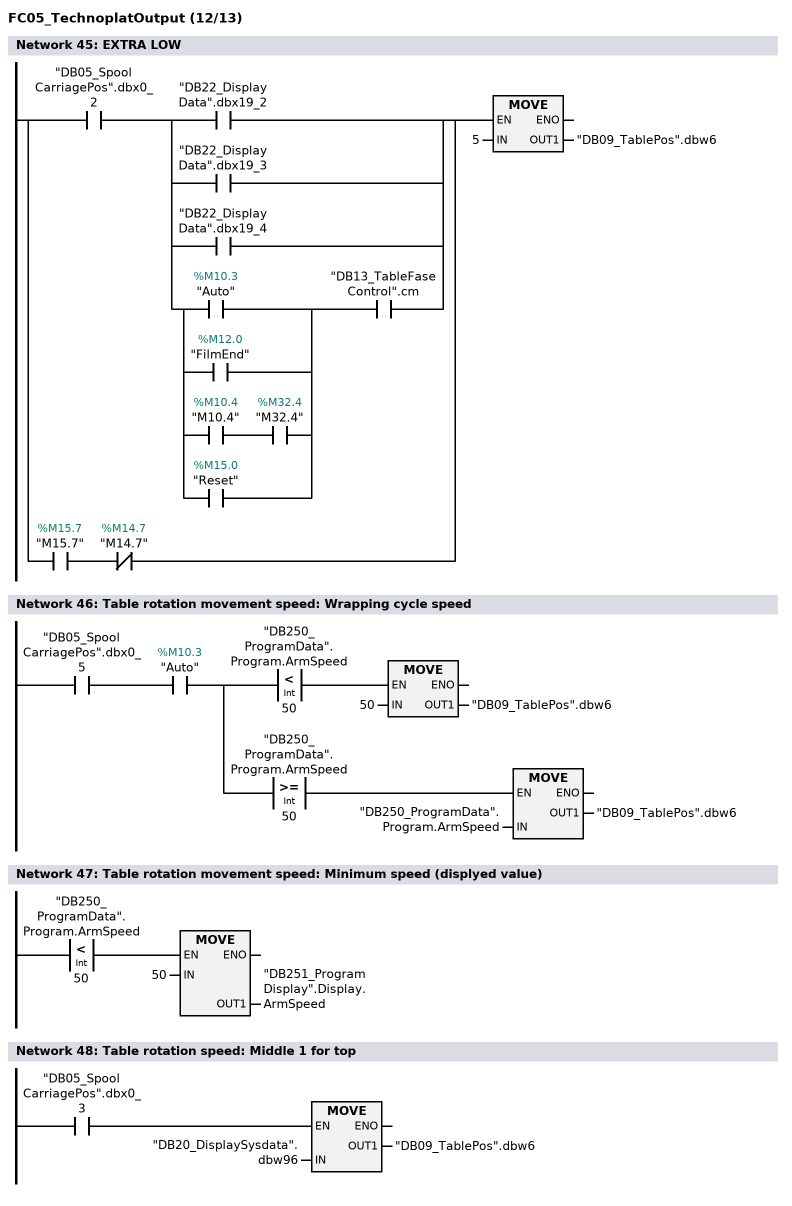
   RUNG wire#powerrail
      Contact( "DB05_SpoolCarriagePos".dbx0_2 )
      wire#w1
      Contact( "DB22_DisplayData".dbx19_2 )
      wire#w2
      { S7_GenerateENO := "TRUE" } Move(in := 5, out1 => "DB09_TablePos".dbw6)
   END_RUNG
   RUNG wire#w1
      Contact( "DB22_DisplayData".dbx19_3 )
   END_RUNG wire#w2
   RUNG wire#w1
      Contact( "DB22_DisplayData".dbx19_4 )
   END_RUNG wire#w2
   RUNG wire#w1
      Contact( "Auto" )
      wire#w3
      Contact( "DB13_TableFaseControl".cm )
   END_RUNG wire#w2
   RUNG wire#w1
      Contact( "FilmEnd" )
   END_RUNG wire#w3
   RUNG wire#w1
      Contact( "M10.4" )
      Contact( "M32.4" )
   END_RUNG wire#w3
   RUNG wire#w1
      Contact( "Reset" )
   END_RUNG wire#w3
   RUNG wire#powerrail
      Contact( "M15.7" )
      I_Contact( "M14.7" )
   END_RUNG wire#w2
   // the same network as SCL:
   IF ("DB05_SpoolCarriagePos".dbx0_2 AND ("DB22_DisplayData".dbx19_2 OR "DB22_DisplayData".dbx19_3 OR "DB22_DisplayData".dbx19_4 OR (("Auto" OR "FilmEnd" OR ("M10.4" AND "M32.4") OR "Reset") AND "DB13_TableFaseControl".cm))) OR ("M15.7" AND NOT "M14.7") THEN
       "DB09_TablePos".dbw6 := 5;
   END_IF;
END_REGION

REGION Network 46: Table rotation movement speed: Wrapping cycle speed
   RUNG wire#powerrail
      Contact( "DB05_SpoolCarriagePos".dbx0_5 )
      Contact( "Auto" )
      wire#w1
      { S7_Templates := "SrcType := Int" } LT_Contact(in1 := "DB250_ProgramData".Program.ArmSpeed, in2 := 50)
      { S7_GenerateENO := "TRUE" } Move(in := 50, out1 => "DB09_TablePos".dbw6)
   END_RUNG
   RUNG wire#w1
      { S7_Templates := "SrcType := Int" } GE_Contact(in1 := "DB250_ProgramData".Program.ArmSpeed, in2 := 50)
      { S7_GenerateENO := "TRUE" } Move(in := "DB250_ProgramData".Program.ArmSpeed, out1 => "DB09_TablePos".dbw6)
   END_RUNG
   // the same network as SCL:
   #_w1 := "DB05_SpoolCarriagePos".dbx0_5 AND "Auto";
   IF #_w1 AND ("DB250_ProgramData".Program.ArmSpeed < 50) THEN "DB09_TablePos".dbw6 := 50; END_IF;
   IF #_w1 AND ("DB250_ProgramData".Program.ArmSpeed >= 50) THEN
       "DB09_TablePos".dbw6 := "DB250_ProgramData".Program.ArmSpeed;
   END_IF;
END_REGION

REGION Network 47: Table rotation movement speed: Minimum speed (displyed value)
   RUNG wire#powerrail
      { S7_Templates := "SrcType := Int" } LT_Contact(in1 := "DB250_ProgramData".Program.ArmSpeed, in2 := 50)
      { S7_GenerateENO := "TRUE" } Move(in := 50, out1 => "DB251_ProgramDisplay".Display.ArmSpeed)
   END_RUNG
   // the same network as SCL:
   IF "DB250_ProgramData".Program.ArmSpeed < 50 THEN "DB251_ProgramDisplay".Display.ArmSpeed := 50; END_IF;
END_REGION

REGION Network 48: Table rotation speed: Middle 1 for top
   RUNG wire#powerrail
      Contact( "DB05_SpoolCarriagePos".dbx0_3 )
      { S7_GenerateENO := "TRUE" } Move(in := "DB20_DisplaySysdata".dbw96, out1 => "DB09_TablePos".dbw6)
   END_RUNG
   // the same network as SCL:
   IF "DB05_SpoolCarriagePos".dbx0_3 THEN "DB09_TablePos".dbw6 := "DB20_DisplaySysdata".dbw96; END_IF;
END_REGION

REGION Network 49: table rotation movement speed range
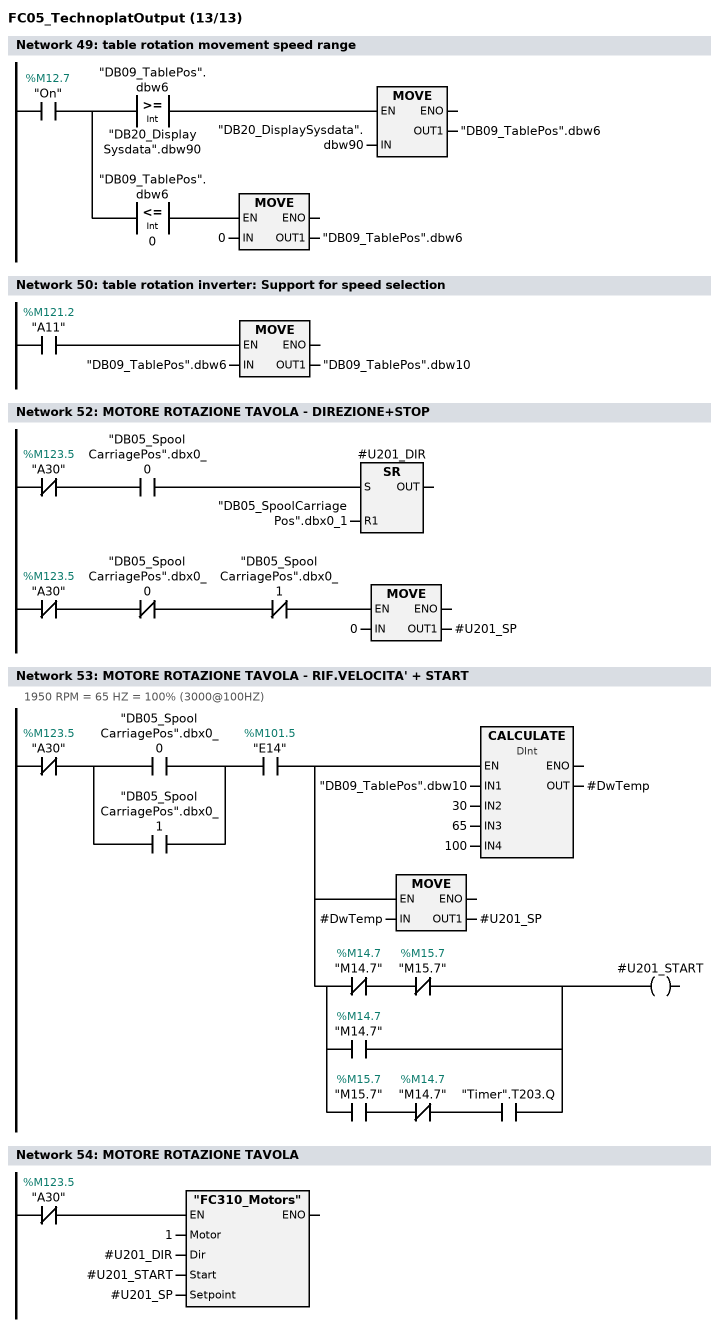
   RUNG wire#powerrail
      Contact( "On" )
      wire#w1
      { S7_Templates := "SrcType := Int" } GE_Contact(in1 := "DB09_TablePos".dbw6, in2 := "DB20_DisplaySysdata".dbw90)
      { S7_GenerateENO := "TRUE" } Move(in := "DB20_DisplaySysdata".dbw90, out1 => "DB09_TablePos".dbw6)
   END_RUNG
   RUNG wire#w1
      { S7_Templates := "SrcType := Int" } LE_Contact(in1 := "DB09_TablePos".dbw6, in2 := 0)
      { S7_GenerateENO := "TRUE" } Move(in := 0, out1 => "DB09_TablePos".dbw6)
   END_RUNG
   // the same network as SCL:
   IF "On" AND ("DB09_TablePos".dbw6 >= "DB20_DisplaySysdata".dbw90) THEN
       "DB09_TablePos".dbw6 := "DB20_DisplaySysdata".dbw90;
   END_IF;
   IF "On" AND ("DB09_TablePos".dbw6 <= 0) THEN "DB09_TablePos".dbw6 := 0; END_IF;
END_REGION

REGION Network 50: table rotation inverter: Support for speed selection
   RUNG wire#powerrail
      Contact( "A11" )
      { S7_GenerateENO := "TRUE" } Move(in := "DB09_TablePos".dbw6, out1 => "DB09_TablePos".dbw10)
   END_RUNG
   // the same network as SCL:
   IF "A11" THEN "DB09_TablePos".dbw10 := "DB09_TablePos".dbw6; END_IF;
END_REGION

REGION Network 51: Table rotation speed conversion
END_REGION

REGION Network 52: MOTORE ROTAZIONE TAVOLA - DIREZIONE+STOP
   RUNG wire#powerrail
      I_Contact( "A30" )
      Contact( "DB05_SpoolCarriagePos".dbx0_0 )
      S_SR(operand := #U201_DIR, r1 := "DB05_SpoolCarriagePos".dbx0_1)
   END_RUNG
   RUNG wire#powerrail
      I_Contact( "A30" )
      I_Contact( "DB05_SpoolCarriagePos".dbx0_0 )
      I_Contact( "DB05_SpoolCarriagePos".dbx0_1 )
      Move(in := 0, out1 => #U201_SP)
   END_RUNG
   // the same network as SCL:
   IF NOT "A30" AND "DB05_SpoolCarriagePos".dbx0_0 THEN
       #U201_DIR := TRUE;   // SR flip-flop
   END_IF;
   IF "DB05_SpoolCarriagePos".dbx0_1 THEN #U201_DIR := FALSE; END_IF;
   IF NOT "A30" AND NOT "DB05_SpoolCarriagePos".dbx0_0 AND NOT "DB05_SpoolCarriagePos".dbx0_1 THEN
       #U201_SP := 0;
   END_IF;
END_REGION

REGION Network 53: MOTORE ROTAZIONE TAVOLA - RIF.VELOCITA' + START
   // 1950 RPM = 65 HZ = 100% (3000@100HZ)
   RUNG wire#powerrail
      I_Contact( "A30" )
      wire#w1
      Contact( "DB05_SpoolCarriagePos".dbx0_0 )
      wire#w2
      Contact( "E14" )
      wire#w3
      { S7_Templates := "SrcType := DInt"; S7_Expression := "(IN1*IN2*IN3)/IN4" } Calculate(in1 := "DB09_TablePos".dbw10, in2 := 30, in3 := 65, in4 := 100, out => #DwTemp)
   END_RUNG
   RUNG wire#w1
      Contact( "DB05_SpoolCarriagePos".dbx0_1 )
   END_RUNG wire#w2
   RUNG wire#w3
      Move(in := #DwTemp, out1 => #U201_SP)
   END_RUNG
   RUNG wire#w3
      I_Contact( "M14.7" )
      I_Contact( "M15.7" )
      wire#w4
      Coil( #U201_START )
   END_RUNG
   RUNG wire#w3
      Contact( "M14.7" )
   END_RUNG wire#w4
   RUNG wire#w3
      Contact( "M15.7" )
      I_Contact( "M14.7" )
      Contact( "Timer".T203.Q )
   END_RUNG wire#w4
   // the same network as SCL:
   #_w1 := NOT "A30" AND ("DB05_SpoolCarriagePos".dbx0_0 OR "DB05_SpoolCarriagePos".dbx0_1) AND "E14";
   IF #_w1 THEN
       #DwTemp := ("DB09_TablePos".dbw10*30*65)/100;
       #U201_SP := #DwTemp;
   END_IF;
   #U201_START := #_w1 AND ((NOT "M14.7" AND NOT "M15.7") OR "M14.7" OR ("M15.7" AND NOT "M14.7" AND "Timer".T203.Q));
END_REGION

REGION Network 54: MOTORE ROTAZIONE TAVOLA
   RUNG wire#powerrail
      I_Contact( "A30" )
      "FC310_Motors"(Motor := 1, Dir := #U201_DIR, Start := #U201_START, Setpoint := #U201_SP)
   END_RUNG
   // the same network as SCL:
   IF NOT "A30" THEN
       "FC310_Motors"(Motor := 1, Dir := #U201_DIR, Start := #U201_START, Setpoint := #U201_SP);
   END_IF;
END_REGION
END_FUNCTION

FUNCTION "FC310_Motors" : Void   // FC310, LAD
{ S7_Optimized_Access := 'TRUE' }
VERSION : 0.1
// stored: AutoNumber false, IsIECCheckEnabled false, SetENOAutomatically false, UDAEnableTagReadback false
   VAR_INPUT
      Motor : Int;   // 0=NO; 1=Arm; 2=Carr; 3=Prestretch; 4=Stretch; 5=SX; 6=CM; 7=DX; 8=Top
      Dir : Bool;   // 0=BKWD; 1=FWD
      Start : Bool;
      Setpoint : Int;
   END_VAR
   VAR_TEMP
      SP_real : Real;
      Carr_Dec_low : DInt;
      Carr_Dec_high : DInt;
   END_VAR
   VAR_TEMP   // added for the SCL form of the ladder/FBD networks
      _w1 : Bool;
      _w2 : Bool;
      _w3 : Bool;
   END_VAR
BEGIN

REGION Network 1: Setpoint conversion
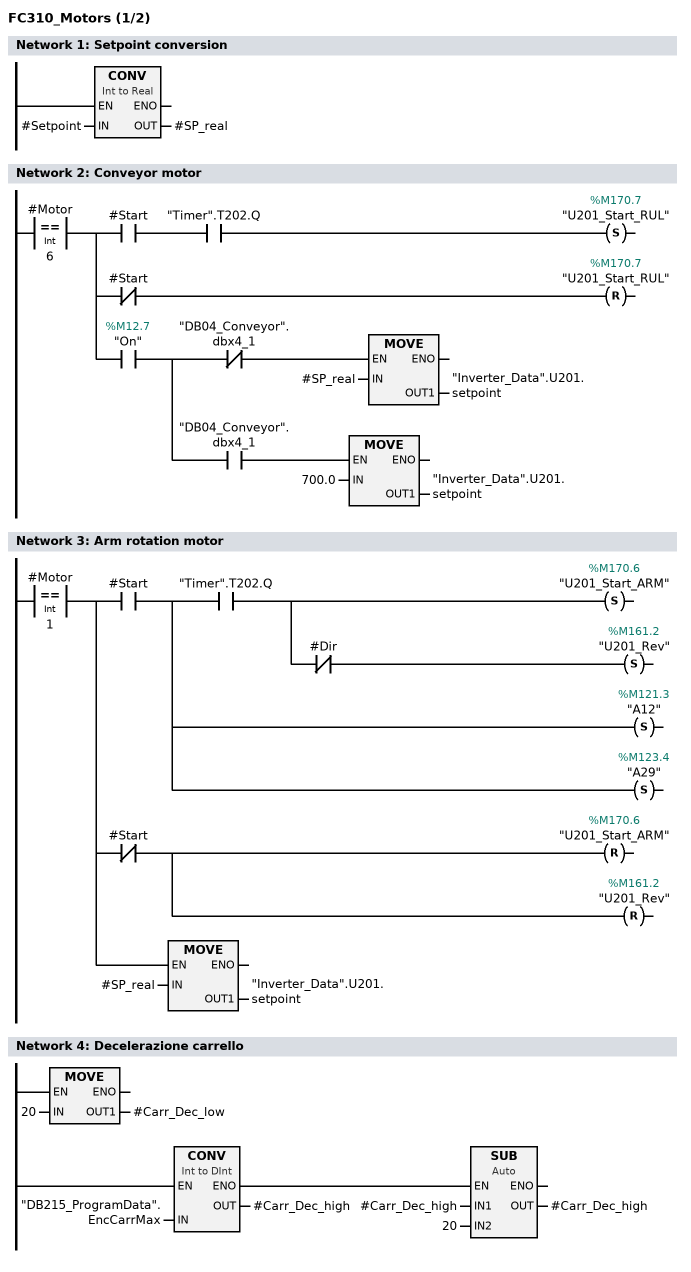
   RUNG wire#powerrail
      { S7_Templates := "[SrcType := Int, DestType := Real]" } Convert(in := #Setpoint, out => #SP_real)
   END_RUNG
   // the same network as SCL:
   #SP_real := INT_TO_REAL(#Setpoint);
END_REGION

REGION Network 2: Conveyor motor
   RUNG wire#powerrail
      { S7_Templates := "SrcType := Int" } EQ_Contact(in1 := #Motor, in2 := 6)
      wire#w1
      Contact( #Start )
      Contact( "Timer".T202.Q )
      S_Coil( "U201_Start_RUL" )
   END_RUNG
   RUNG wire#w1
      I_Contact( #Start )
      R_Coil( "U201_Start_RUL" )
   END_RUNG
   RUNG wire#w1
      Contact( "On" )
      wire#w2
      I_Contact( "DB04_Conveyor".dbx4_1 )
      Move(in := #SP_real, out1 => "Inverter_Data".U201.setpoint)
   END_RUNG
   RUNG wire#w2
      Contact( "DB04_Conveyor".dbx4_1 )
      Move(in := 700.0, out1 => "Inverter_Data".U201.setpoint)
   END_RUNG
   // the same network as SCL:
   #_w1 := #Motor = 6;
   IF #_w1 AND #Start AND "Timer".T202.Q THEN "U201_Start_RUL" := TRUE; END_IF;
   IF #_w1 AND NOT #Start THEN "U201_Start_RUL" := FALSE; END_IF;
   #_w2 := #_w1 AND "On";
   IF #_w2 AND NOT "DB04_Conveyor".dbx4_1 THEN "Inverter_Data".U201.setpoint := #SP_real; END_IF;
   IF #_w2 AND "DB04_Conveyor".dbx4_1 THEN "Inverter_Data".U201.setpoint := 700.0; END_IF;
END_REGION

REGION Network 3: Arm rotation motor
   RUNG wire#powerrail
      { S7_Templates := "SrcType := Int" } EQ_Contact(in1 := #Motor, in2 := 1)
      wire#w1
      Contact( #Start )
      wire#w2
      Contact( "Timer".T202.Q )
      wire#w3
      S_Coil( "U201_Start_ARM" )
   END_RUNG
   RUNG wire#w3
      I_Contact( #Dir )
      S_Coil( "U201_Rev" )
   END_RUNG
   RUNG wire#w2
      S_Coil( "A12" )
   END_RUNG
   RUNG wire#w2
      S_Coil( "A29" )
   END_RUNG
   RUNG wire#w1
      I_Contact( #Start )
      wire#w4
      R_Coil( "U201_Start_ARM" )
   END_RUNG
   RUNG wire#w4
      R_Coil( "U201_Rev" )
   END_RUNG
   RUNG wire#w1
      Move(in := #SP_real, out1 => "Inverter_Data".U201.setpoint)
   END_RUNG
   // the same network as SCL:
   #_w1 := #Motor = 1;
   #_w2 := #_w1 AND #Start;
   #_w3 := #_w2 AND "Timer".T202.Q;
   IF #_w3 THEN "U201_Start_ARM" := TRUE; END_IF;
   IF #_w3 AND NOT #Dir THEN "U201_Rev" := TRUE; END_IF;
   IF #_w2 THEN
       "A12" := TRUE;
       "A29" := TRUE;
   END_IF;
   IF #_w1 AND NOT #Start THEN
       "U201_Start_ARM" := FALSE;
       "U201_Rev" := FALSE;
   END_IF;
   IF #_w1 THEN "Inverter_Data".U201.setpoint := #SP_real; END_IF;
END_REGION

REGION Network 4: Decelerazione carrello
   RUNG wire#powerrail
      Move(in := 20, out1 => #Carr_Dec_low)
   END_RUNG
   RUNG wire#powerrail
      { S7_Templates := "[SrcType := Int, DestType := DInt]" } Convert(in := "DB215_ProgramData".EncCarrMax, out => #Carr_Dec_high)
      Sub(in1 := #Carr_Dec_high, in2 := 20, out => #Carr_Dec_high)
   END_RUNG
   // the same network as SCL:
   #Carr_Dec_low := 20;
   #Carr_Dec_high := INT_TO_DINT("DB215_ProgramData".EncCarrMax);
   #Carr_Dec_high := #Carr_Dec_high - 20;
END_REGION

REGION Network 5: Carriage motor
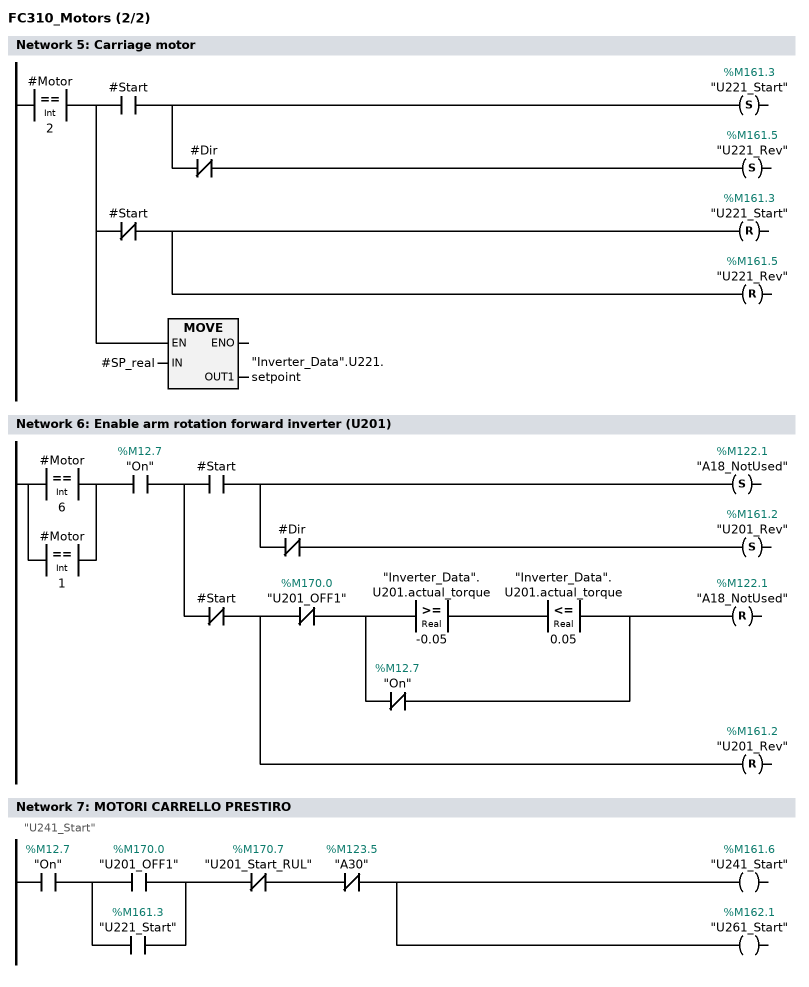
   RUNG wire#powerrail
      { S7_Templates := "SrcType := Int" } EQ_Contact(in1 := #Motor, in2 := 2)
      wire#w1
      Contact( #Start )
      wire#w2
      S_Coil( "U221_Start" )
   END_RUNG
   RUNG wire#w2
      I_Contact( #Dir )
      S_Coil( "U221_Rev" )
   END_RUNG
   RUNG wire#w1
      I_Contact( #Start )
      wire#w3
      R_Coil( "U221_Start" )
   END_RUNG
   RUNG wire#w3
      R_Coil( "U221_Rev" )
   END_RUNG
   RUNG wire#w1
      Move(in := #SP_real, out1 => "Inverter_Data".U221.setpoint)
   END_RUNG
   // the same network as SCL:
   #_w1 := #Motor = 2;
   #_w2 := #_w1 AND #Start;
   IF #_w2 THEN "U221_Start" := TRUE; END_IF;
   IF #_w2 AND NOT #Dir THEN "U221_Rev" := TRUE; END_IF;
   IF #_w1 AND NOT #Start THEN
       "U221_Start" := FALSE;
       "U221_Rev" := FALSE;
   END_IF;
   IF #_w1 THEN "Inverter_Data".U221.setpoint := #SP_real; END_IF;
END_REGION

REGION Network 6: Enable arm rotation forward inverter (U201)
   RUNG wire#powerrail
      { S7_Templates := "SrcType := Int" } EQ_Contact(in1 := #Motor, in2 := 6)
      wire#w1
      Contact( "On" )
      wire#w2
      Contact( #Start )
      wire#w3
      S_Coil( "A18_NotUsed" )
   END_RUNG
   RUNG wire#powerrail
      { S7_Templates := "SrcType := Int" } EQ_Contact(in1 := #Motor, in2 := 1)
   END_RUNG wire#w1
   RUNG wire#w3
      I_Contact( #Dir )
      S_Coil( "U201_Rev" )
   END_RUNG
   RUNG wire#w2
      I_Contact( #Start )
      wire#w4
      I_Contact( "U201_OFF1" )
      wire#w5
      { S7_Templates := "SrcType := Real" } GE_Contact(in1 := "Inverter_Data".U201.actual_torque, in2 := -0.05)
      { S7_Templates := "SrcType := Real" } LE_Contact(in1 := "Inverter_Data".U201.actual_torque, in2 := 0.05)
      wire#w6
      R_Coil( "A18_NotUsed" )
   END_RUNG
   RUNG wire#w5
      I_Contact( "On" )
   END_RUNG wire#w6
   RUNG wire#w4
      R_Coil( "U201_Rev" )
   END_RUNG
   // the same network as SCL:
   #_w1 := ((#Motor = 6) OR (#Motor = 1)) AND "On";
   #_w2 := #_w1 AND #Start;
   IF #_w2 THEN "A18_NotUsed" := TRUE; END_IF;
   IF #_w2 AND NOT #Dir THEN "U201_Rev" := TRUE; END_IF;
   #_w3 := #_w1 AND NOT #Start;
   IF #_w3 AND NOT "U201_OFF1" AND ((("Inverter_Data".U201.actual_torque >= (-0.05)) AND ("Inverter_Data".U201.actual_torque <= 0.05)) OR NOT "On") THEN
       "A18_NotUsed" := FALSE;
   END_IF;
   IF #_w3 THEN "U201_Rev" := FALSE; END_IF;
END_REGION

REGION Network 7: MOTORI CARRELLO PRESTIRO
   // "U241_Start"
   RUNG wire#powerrail
      Contact( "On" )
      wire#w1
      Contact( "U201_OFF1" )
      wire#w2
      I_Contact( "U201_Start_RUL" )
      I_Contact( "A30" )
      wire#w3
      Coil( "U241_Start" )
   END_RUNG
   RUNG wire#w1
      Contact( "U221_Start" )
   END_RUNG wire#w2
   RUNG wire#w3
      Coil( "U261_Start" )
   END_RUNG
   // the same network as SCL:
   "U241_Start" := "On" AND ("U201_OFF1" OR "U221_Start") AND NOT "U201_Start_RUL" AND NOT "A30";
   "U261_Start" := "U241_Start";
END_REGION
END_FUNCTION

FUNCTION "FC04_TechnoplatAlarm" : Void   // FC4, LAD
TITLE = Alarm for the machine
{ S7_Optimized_Access := 'FALSE' }
AUTHOR : Robopac
VERSION : 0.0
// stored: AutoNumber false, IsIECCheckEnabled false, SetENOAutomatically false, UDAEnableTagReadback false
BEGIN

REGION Network 1: Alarm 1: Pressure switch (Technoplat)
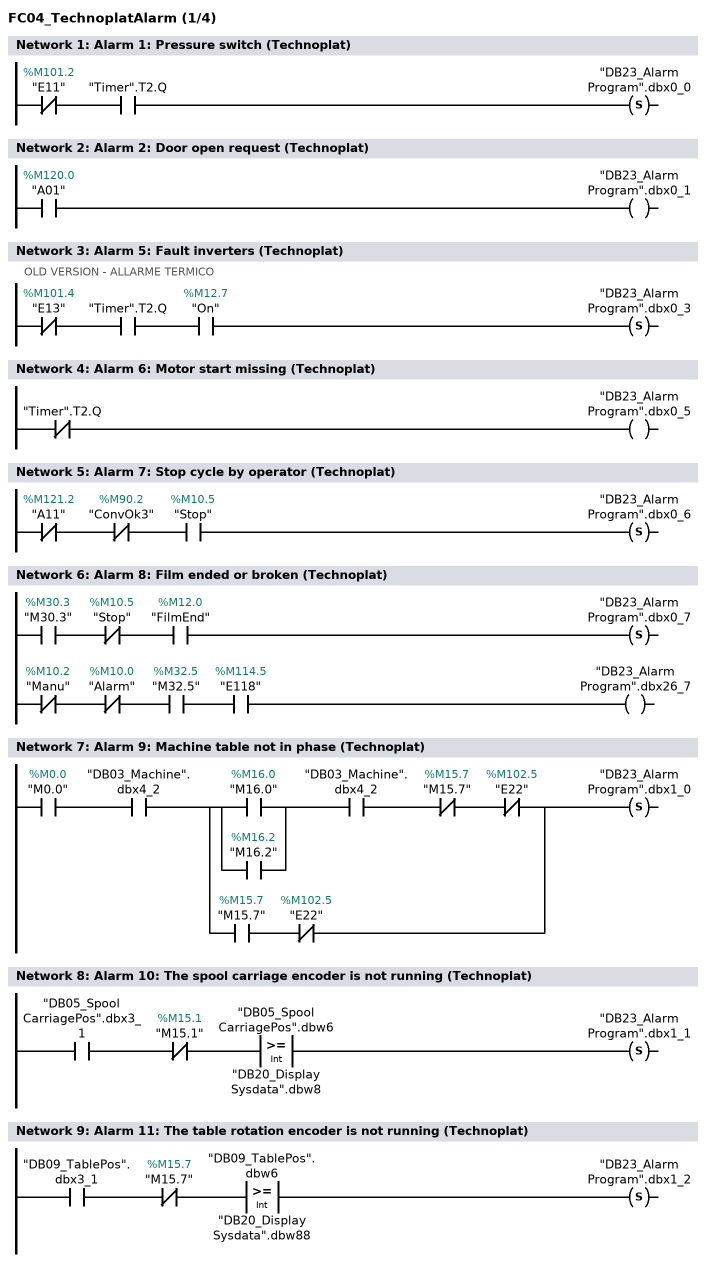
   RUNG wire#powerrail
      I_Contact( "E11" )
      Contact( "Timer".T2.Q )
      S_Coil( "DB23_AlarmProgram".dbx0_0 )
   END_RUNG
   // the same network as SCL:
   IF NOT "E11" AND "Timer".T2.Q THEN "DB23_AlarmProgram".dbx0_0 := TRUE; END_IF;
END_REGION

REGION Network 2: Alarm 2: Door open request (Technoplat)
   RUNG wire#powerrail
      Contact( "A01" )
      Coil( "DB23_AlarmProgram".dbx0_1 )
   END_RUNG
   // the same network as SCL:
   "DB23_AlarmProgram".dbx0_1 := "A01";
END_REGION

REGION Network 3: Alarm 5: Fault inverters (Technoplat)
   // OLD VERSION - ALLARME TERMICO
   RUNG wire#powerrail
      I_Contact( "E13" )
      Contact( "Timer".T2.Q )
      Contact( "On" )
      S_Coil( "DB23_AlarmProgram".dbx0_3 )
   END_RUNG
   // the same network as SCL:
   IF NOT "E13" AND "Timer".T2.Q AND "On" THEN "DB23_AlarmProgram".dbx0_3 := TRUE; END_IF;
END_REGION

REGION Network 4: Alarm 6: Motor start missing (Technoplat)
   RUNG wire#powerrail
      I_Contact( "Timer".T2.Q )
      Coil( "DB23_AlarmProgram".dbx0_5 )
   END_RUNG
   // the same network as SCL:
   "DB23_AlarmProgram".dbx0_5 := NOT "Timer".T2.Q;
END_REGION

REGION Network 5: Alarm 7: Stop cycle by operator (Technoplat)
   RUNG wire#powerrail
      I_Contact( "A11" )
      I_Contact( "ConvOk3" )
      Contact( "Stop" )
      S_Coil( "DB23_AlarmProgram".dbx0_6 )
   END_RUNG
   // the same network as SCL:
   IF NOT "A11" AND NOT "ConvOk3" AND "Stop" THEN "DB23_AlarmProgram".dbx0_6 := TRUE; END_IF;
END_REGION

REGION Network 6: Alarm 8: Film ended or broken (Technoplat)
   RUNG wire#powerrail
      Contact( "M30.3" )
      I_Contact( "Stop" )
      Contact( "FilmEnd" )
      S_Coil( "DB23_AlarmProgram".dbx0_7 )
   END_RUNG
   RUNG wire#powerrail
      I_Contact( "Manu" )
      I_Contact( "Alarm" )
      Contact( "M32.5" )
      Contact( "E118" )
      Coil( "DB23_AlarmProgram".dbx26_7 )
   END_RUNG
   // the same network as SCL:
   IF "M30.3" AND NOT "Stop" AND "FilmEnd" THEN "DB23_AlarmProgram".dbx0_7 := TRUE; END_IF;
   "DB23_AlarmProgram".dbx26_7 := NOT "Manu" AND NOT "Alarm" AND "M32.5" AND "E118";
END_REGION

REGION Network 7: Alarm 9: Machine table not in phase (Technoplat)
   RUNG wire#powerrail
      Contact( "M0.0" )
      Contact( "DB03_Machine".dbx4_2 )
      wire#w1
      Contact( "M16.0" )
      wire#w2
      Contact( "DB03_Machine".dbx4_2 )
      I_Contact( "M15.7" )
      I_Contact( "E22" )
      wire#w3
      S_Coil( "DB23_AlarmProgram".dbx1_0 )
   END_RUNG
   RUNG wire#w1
      Contact( "M16.2" )
   END_RUNG wire#w2
   RUNG wire#w1
      Contact( "M15.7" )
      I_Contact( "E22" )
   END_RUNG wire#w3
   // the same network as SCL:
   IF "M0.0" AND "DB03_Machine".dbx4_2 AND ((("M16.0" OR "M16.2") AND "DB03_Machine".dbx4_2 AND NOT "M15.7" AND NOT "E22") OR ("M15.7" AND NOT "E22")) THEN
       "DB23_AlarmProgram".dbx1_0 := TRUE;
   END_IF;
END_REGION

REGION Network 8: Alarm 10: The spool carriage encoder is not running (Technoplat)
   RUNG wire#powerrail
      Contact( "DB05_SpoolCarriagePos".dbx3_1 )
      I_Contact( "M15.1" )
      { S7_Templates := "SrcType := Int" } GE_Contact(in1 := "DB05_SpoolCarriagePos".dbw6, in2 := "DB20_DisplaySysdata".dbw8)
      S_Coil( "DB23_AlarmProgram".dbx1_1 )
   END_RUNG
   // the same network as SCL:
   IF "DB05_SpoolCarriagePos".dbx3_1 AND NOT "M15.1" AND ("DB05_SpoolCarriagePos".dbw6 >= "DB20_DisplaySysdata".dbw8) THEN
       "DB23_AlarmProgram".dbx1_1 := TRUE;
   END_IF;
END_REGION

REGION Network 9: Alarm 11: The table rotation encoder is not running (Technoplat)
   RUNG wire#powerrail
      Contact( "DB09_TablePos".dbx3_1 )
      I_Contact( "M15.7" )
      { S7_Templates := "SrcType := Int" } GE_Contact(in1 := "DB09_TablePos".dbw6, in2 := "DB20_DisplaySysdata".dbw88)
      S_Coil( "DB23_AlarmProgram".dbx1_2 )
   END_RUNG
   // the same network as SCL:
   IF "DB09_TablePos".dbx3_1 AND NOT "M15.7" AND ("DB09_TablePos".dbw6 >= "DB20_DisplaySysdata".dbw88) THEN
       "DB23_AlarmProgram".dbx1_2 := TRUE;
   END_IF;
END_REGION

REGION Network 10: Alarm 12: Overspeed for arm rotation (Technoplat)
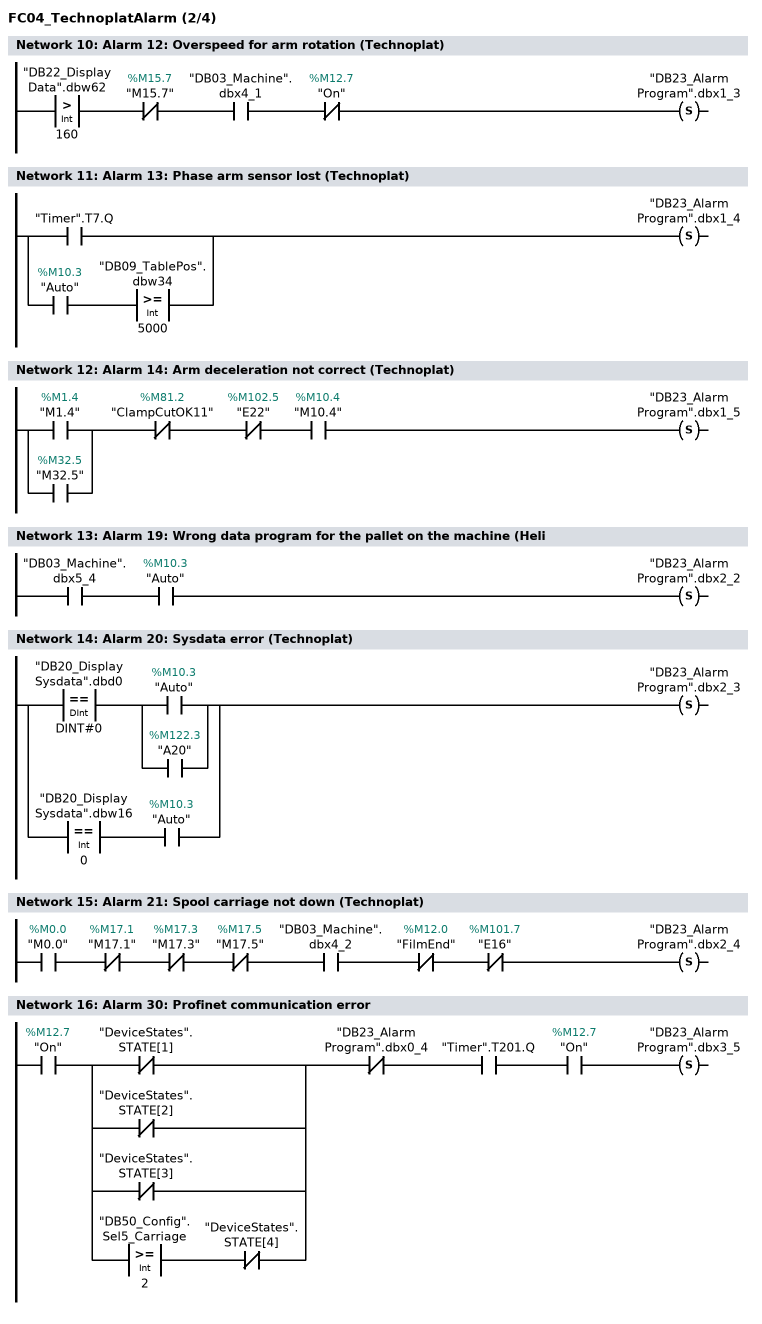
   RUNG wire#powerrail
      { S7_Templates := "SrcType := Int" } GT_Contact(in1 := "DB22_DisplayData".dbw62, in2 := 160)
      I_Contact( "M15.7" )
      Contact( "DB03_Machine".dbx4_1 )
      I_Contact( "On" )
      S_Coil( "DB23_AlarmProgram".dbx1_3 )
   END_RUNG
   // the same network as SCL:
   IF ("DB22_DisplayData".dbw62 > 160) AND NOT "M15.7" AND "DB03_Machine".dbx4_1 AND NOT "On" THEN
       "DB23_AlarmProgram".dbx1_3 := TRUE;
   END_IF;
END_REGION

REGION Network 11: Alarm 13: Phase arm sensor lost (Technoplat)
   RUNG wire#powerrail
      Contact( "Timer".T7.Q )
      wire#w1
      S_Coil( "DB23_AlarmProgram".dbx1_4 )
   END_RUNG
   RUNG wire#powerrail
      Contact( "Auto" )
      { S7_Templates := "SrcType := Int" } GE_Contact(in1 := "DB09_TablePos".dbw34, in2 := 5000)
   END_RUNG wire#w1
   // the same network as SCL:
   IF "Timer".T7.Q OR ("Auto" AND ("DB09_TablePos".dbw34 >= 5000)) THEN
       "DB23_AlarmProgram".dbx1_4 := TRUE;
   END_IF;
END_REGION

REGION Network 12: Alarm 14: Arm deceleration not correct (Technoplat)
   RUNG wire#powerrail
      Contact( "M1.4" )
      wire#w1
      I_Contact( "ClampCutOK11" )
      I_Contact( "E22" )
      Contact( "M10.4" )
      S_Coil( "DB23_AlarmProgram".dbx1_5 )
   END_RUNG
   RUNG wire#powerrail
      Contact( "M32.5" )
   END_RUNG wire#w1
   // the same network as SCL:
   IF ("M1.4" OR "M32.5") AND NOT "ClampCutOK11" AND NOT "E22" AND "M10.4" THEN
       "DB23_AlarmProgram".dbx1_5 := TRUE;
   END_IF;
END_REGION

REGION Network 13: Alarm 19: Wrong data program for the pallet on the machine (Heli
   RUNG wire#powerrail
      Contact( "DB03_Machine".dbx5_4 )
      Contact( "Auto" )
      S_Coil( "DB23_AlarmProgram".dbx2_2 )
   END_RUNG
   // the same network as SCL:
   IF "DB03_Machine".dbx5_4 AND "Auto" THEN "DB23_AlarmProgram".dbx2_2 := TRUE; END_IF;
END_REGION

REGION Network 14: Alarm 20: Sysdata error (Technoplat)
   RUNG wire#powerrail
      { S7_Templates := "SrcType := DInt" } EQ_Contact(in1 := "DB20_DisplaySysdata".dbd0, in2 := DINT#0)
      wire#w1
      Contact( "Auto" )
      wire#w2
      S_Coil( "DB23_AlarmProgram".dbx2_3 )
   END_RUNG
   RUNG wire#w1
      Contact( "A20" )
   END_RUNG wire#w2
   RUNG wire#powerrail
      { S7_Templates := "SrcType := Int" } EQ_Contact(in1 := "DB20_DisplaySysdata".dbw16, in2 := 0)
      Contact( "Auto" )
   END_RUNG wire#w2
   // the same network as SCL:
   IF (("DB20_DisplaySysdata".dbd0 = DINT#0) AND ("Auto" OR "A20")) OR (("DB20_DisplaySysdata".dbw16 = 0) AND "Auto") THEN
       "DB23_AlarmProgram".dbx2_3 := TRUE;
   END_IF;
END_REGION

REGION Network 15: Alarm 21: Spool carriage not down (Technoplat)
   RUNG wire#powerrail
      Contact( "M0.0" )
      I_Contact( "M17.1" )
      I_Contact( "M17.3" )
      I_Contact( "M17.5" )
      Contact( "DB03_Machine".dbx4_2 )
      I_Contact( "FilmEnd" )
      I_Contact( "E16" )
      S_Coil( "DB23_AlarmProgram".dbx2_4 )
   END_RUNG
   // the same network as SCL:
   IF "M0.0" AND NOT "M17.1" AND NOT "M17.3" AND NOT "M17.5" AND "DB03_Machine".dbx4_2 AND NOT "FilmEnd" AND NOT "E16" THEN
       "DB23_AlarmProgram".dbx2_4 := TRUE;
   END_IF;
END_REGION

REGION Network 16: Alarm 30: Profinet communication error
   RUNG wire#powerrail
      Contact( "On" )
      wire#w1
      I_Contact( "DeviceStates".STATE[1] )
      wire#w2
      I_Contact( "DB23_AlarmProgram".dbx0_4 )
      Contact( "Timer".T201.Q )
      Contact( "On" )
      S_Coil( "DB23_AlarmProgram".dbx3_5 )
   END_RUNG
   RUNG wire#w1
      I_Contact( "DeviceStates".STATE[2] )
   END_RUNG wire#w2
   RUNG wire#w1
      I_Contact( "DeviceStates".STATE[3] )
   END_RUNG wire#w2
   RUNG wire#w1
      { S7_Templates := "SrcType := Int" } GE_Contact(in1 := "DB50_Config".Sel5_Carriage, in2 := 2)
      I_Contact( "DeviceStates".STATE[4] )
   END_RUNG wire#w2
   // the same network as SCL:
   IF "On" AND (NOT "DeviceStates".STATE[1] OR NOT "DeviceStates".STATE[2] OR NOT "DeviceStates".STATE[3] OR (("DB50_Config".Sel5_Carriage >= 2) AND NOT "DeviceStates".STATE[4])) AND NOT "DB23_AlarmProgram".dbx0_4 AND "Timer".T201.Q AND "On" THEN
       "DB23_AlarmProgram".dbx3_5 := TRUE;
   END_IF;
END_REGION

REGION Network 17: Alarm 31: Modbus communication error
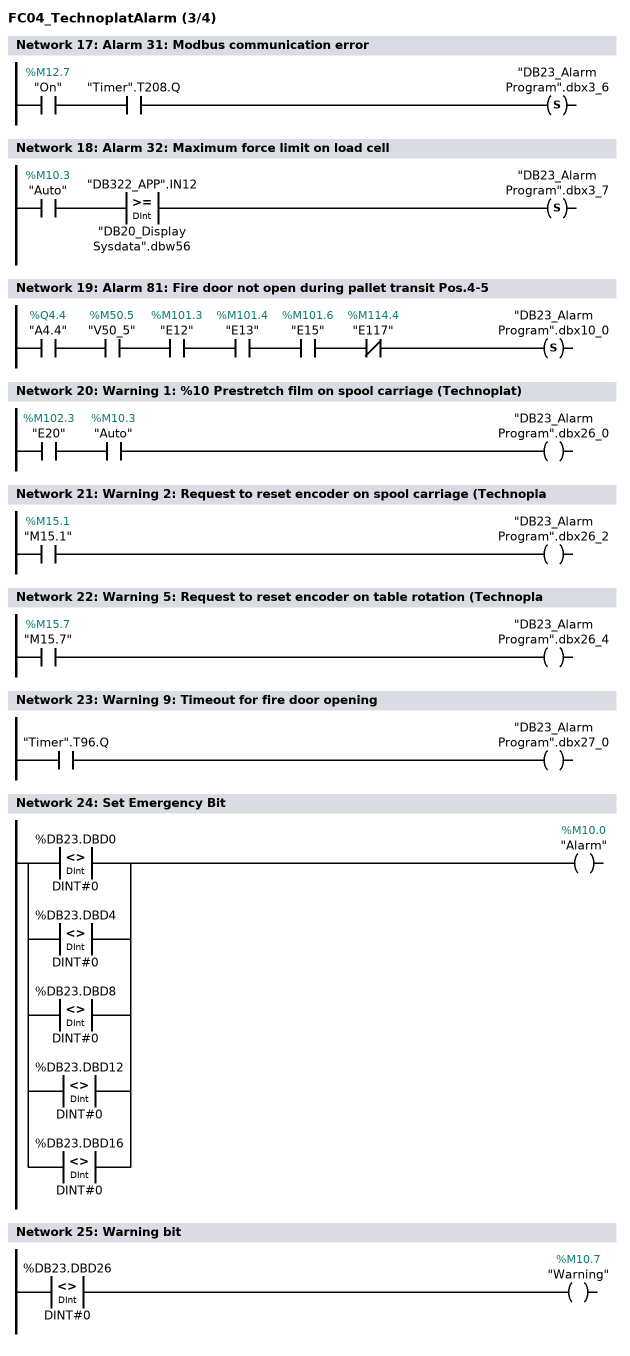
   RUNG wire#powerrail
      Contact( "On" )
      Contact( "Timer".T208.Q )
      S_Coil( "DB23_AlarmProgram".dbx3_6 )
   END_RUNG
   // the same network as SCL:
   IF "On" AND "Timer".T208.Q THEN "DB23_AlarmProgram".dbx3_6 := TRUE; END_IF;
END_REGION

REGION Network 18: Alarm 32: Maximum force limit on load cell
   RUNG wire#powerrail
      Contact( "Auto" )
      { S7_Templates := "SrcType := DInt" } GE_Contact(in1 := "DB322_APP".IN12, in2 := "DB20_DisplaySysdata".dbw56)
      S_Coil( "DB23_AlarmProgram".dbx3_7 )
   END_RUNG
   // the same network as SCL:
   IF "Auto" AND ("DB322_APP".IN12 >= "DB20_DisplaySysdata".dbw56) THEN
       "DB23_AlarmProgram".dbx3_7 := TRUE;
   END_IF;
END_REGION

REGION Network 19: Alarm 81: Fire door not open during pallet transit Pos.4-5
   RUNG wire#powerrail
      Contact( "A4.4" )
      Contact( "V50_5" )
      Contact( "E12" )
      Contact( "E13" )
      Contact( "E15" )
      I_Contact( "E117" )
      S_Coil( "DB23_AlarmProgram".dbx10_0 )
   END_RUNG
   // the same network as SCL:
   IF "A4.4" AND "V50_5" AND "E12" AND "E13" AND "E15" AND NOT "E117" THEN
       "DB23_AlarmProgram".dbx10_0 := TRUE;
   END_IF;
END_REGION

REGION Network 20: Warning 1: %10 Prestretch film on spool carriage (Technoplat)
   RUNG wire#powerrail
      Contact( "E20" )
      Contact( "Auto" )
      Coil( "DB23_AlarmProgram".dbx26_0 )
   END_RUNG
   // the same network as SCL:
   "DB23_AlarmProgram".dbx26_0 := "E20" AND "Auto";
END_REGION

REGION Network 21: Warning 2: Request to reset encoder on spool carriage (Technopla
   RUNG wire#powerrail
      Contact( "M15.1" )
      Coil( "DB23_AlarmProgram".dbx26_2 )
   END_RUNG
   // the same network as SCL:
   "DB23_AlarmProgram".dbx26_2 := "M15.1";
END_REGION

REGION Network 22: Warning 5: Request to reset encoder on table rotation (Technopla
   RUNG wire#powerrail
      Contact( "M15.7" )
      Coil( "DB23_AlarmProgram".dbx26_4 )
   END_RUNG
   // the same network as SCL:
   "DB23_AlarmProgram".dbx26_4 := "M15.7";
END_REGION

REGION Network 23: Warning 9: Timeout for fire door opening
   RUNG wire#powerrail
      Contact( "Timer".T96.Q )
      Coil( "DB23_AlarmProgram".dbx27_0 )
   END_RUNG
   // the same network as SCL:
   "DB23_AlarmProgram".dbx27_0 := "Timer".T96.Q;
END_REGION

REGION Network 24: Set Emergency Bit
   RUNG wire#powerrail
      { S7_Templates := "SrcType := DInt" } NE_Contact(in1 := %DB23.DBD0, in2 := DINT#0)
      wire#w1
      Coil( "Alarm" )
   END_RUNG
   RUNG wire#powerrail
      { S7_Templates := "SrcType := DInt" } NE_Contact(in1 := %DB23.DBD4, in2 := DINT#0)
   END_RUNG wire#w1
   RUNG wire#powerrail
      { S7_Templates := "SrcType := DInt" } NE_Contact(in1 := %DB23.DBD8, in2 := DINT#0)
   END_RUNG wire#w1
   RUNG wire#powerrail
      { S7_Templates := "SrcType := DInt" } NE_Contact(in1 := %DB23.DBD12, in2 := DINT#0)
   END_RUNG wire#w1
   RUNG wire#powerrail
      { S7_Templates := "SrcType := DInt" } NE_Contact(in1 := %DB23.DBD16, in2 := DINT#0)
   END_RUNG wire#w1
   // the same network as SCL:
   "Alarm" := (%DB23.DBD0 <> DINT#0) OR (%DB23.DBD4 <> DINT#0) OR (%DB23.DBD8 <> DINT#0) OR (%DB23.DBD12 <> DINT#0) OR (%DB23.DBD16 <> DINT#0);
END_REGION

REGION Network 25: Warning bit
   RUNG wire#powerrail
      { S7_Templates := "SrcType := DInt" } NE_Contact(in1 := %DB23.DBD26, in2 := DINT#0)
      Coil( "Warning" )
   END_RUNG
   // the same network as SCL:
   "Warning" := %DB23.DBD26 <> DINT#0;
END_REGION

REGION Network 26: First cycle
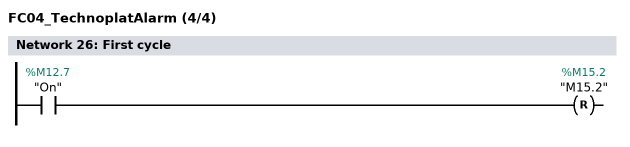
   RUNG wire#powerrail
      Contact( "On" )
      R_Coil( "M15.2" )
   END_RUNG
   // the same network as SCL:
   IF "On" THEN "M15.2" := FALSE; END_IF;
END_REGION
END_FUNCTION

FUNCTION "FC01_SupportOut" : Void   // FC1, LAD
TITLE = Output support memory
{ S7_Optimized_Access := 'FALSE' }
AUTHOR : Robopac
VERSION : 0.0
// stored: AutoNumber false, IsIECCheckEnabled false, SetENOAutomatically false, UDAEnableTagReadback false
BEGIN

REGION Network 1: STANDARD
END_REGION

REGION Network 2: Emergency mode lamp (Technoplat)
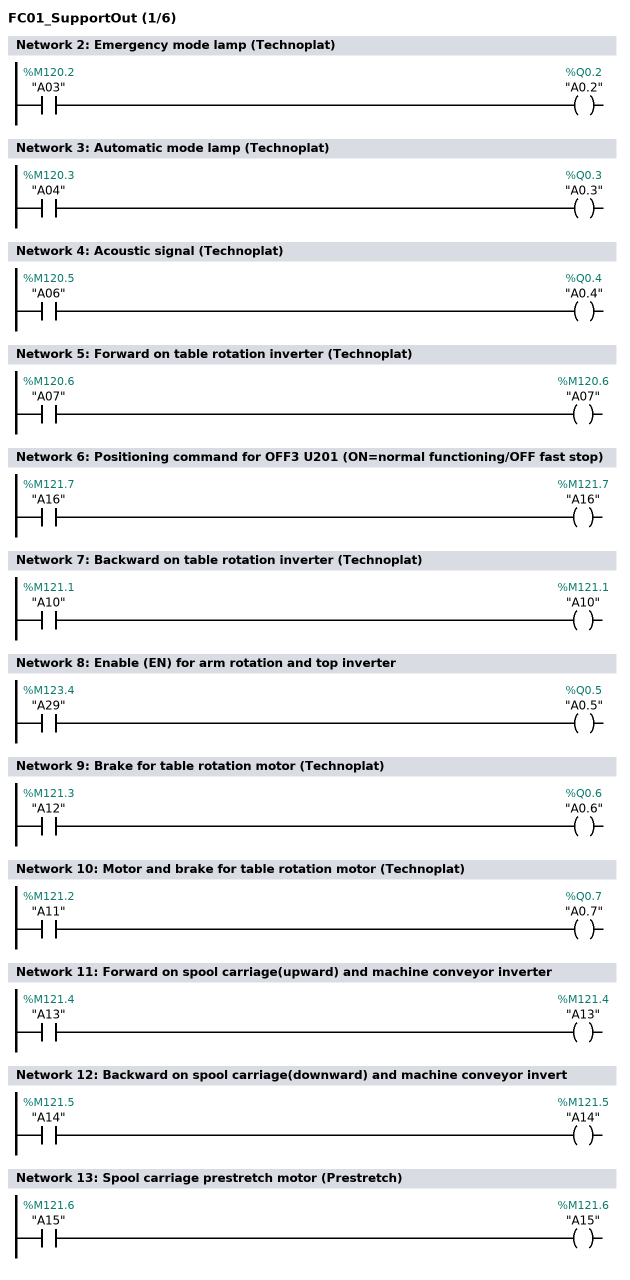
   RUNG wire#powerrail
      Contact( "A03" )
      Coil( "A0.2" )
   END_RUNG
   // the same network as SCL:
   "A0.2" := "A03";
END_REGION

REGION Network 3: Automatic mode lamp (Technoplat)
   RUNG wire#powerrail
      Contact( "A04" )
      Coil( "A0.3" )
   END_RUNG
   // the same network as SCL:
   "A0.3" := "A04";
END_REGION

REGION Network 4: Acoustic signal (Technoplat)
   RUNG wire#powerrail
      Contact( "A06" )
      Coil( "A0.4" )
   END_RUNG
   // the same network as SCL:
   "A0.4" := "A06";
END_REGION

REGION Network 5: Forward on table rotation inverter (Technoplat)
   RUNG wire#powerrail
      Contact( "A07" )
      Coil( "A07" )
   END_RUNG
   // the same network as SCL:
   "A07" := "A07";
END_REGION

REGION Network 6: Positioning command for OFF3 U201 (ON=normal functioning/OFF fast stop)
   RUNG wire#powerrail
      Contact( "A16" )
      Coil( "A16" )
   END_RUNG
   // the same network as SCL:
   "A16" := "A16";
END_REGION

REGION Network 7: Backward on table rotation inverter (Technoplat)
   RUNG wire#powerrail
      Contact( "A10" )
      Coil( "A10" )
   END_RUNG
   // the same network as SCL:
   "A10" := "A10";
END_REGION

REGION Network 8: Enable (EN) for arm rotation and top inverter
   RUNG wire#powerrail
      Contact( "A29" )
      Coil( "A0.5" )
   END_RUNG
   // the same network as SCL:
   "A0.5" := "A29";
END_REGION

REGION Network 9: Brake for table rotation motor (Technoplat)
   RUNG wire#powerrail
      Contact( "A12" )
      Coil( "A0.6" )
   END_RUNG
   // the same network as SCL:
   "A0.6" := "A12";
END_REGION

REGION Network 10: Motor and brake for table rotation motor (Technoplat)
   RUNG wire#powerrail
      Contact( "A11" )
      Coil( "A0.7" )
   END_RUNG
   // the same network as SCL:
   "A0.7" := "A11";
END_REGION

REGION Network 11: Forward on spool carriage(upward) and machine conveyor inverter
   RUNG wire#powerrail
      Contact( "A13" )
      Coil( "A13" )
   END_RUNG
   // the same network as SCL:
   "A13" := "A13";
END_REGION

REGION Network 12: Backward on spool carriage(downward) and machine conveyor invert
   RUNG wire#powerrail
      Contact( "A14" )
      Coil( "A14" )
   END_RUNG
   // the same network as SCL:
   "A14" := "A14";
END_REGION

REGION Network 13: Spool carriage prestretch motor (Prestretch)
   RUNG wire#powerrail
      Contact( "A15" )
      Coil( "A15" )
   END_RUNG
   // the same network as SCL:
   "A15" := "A15";
END_REGION

REGION Network 14: Film clamp opening (Claw clamp)
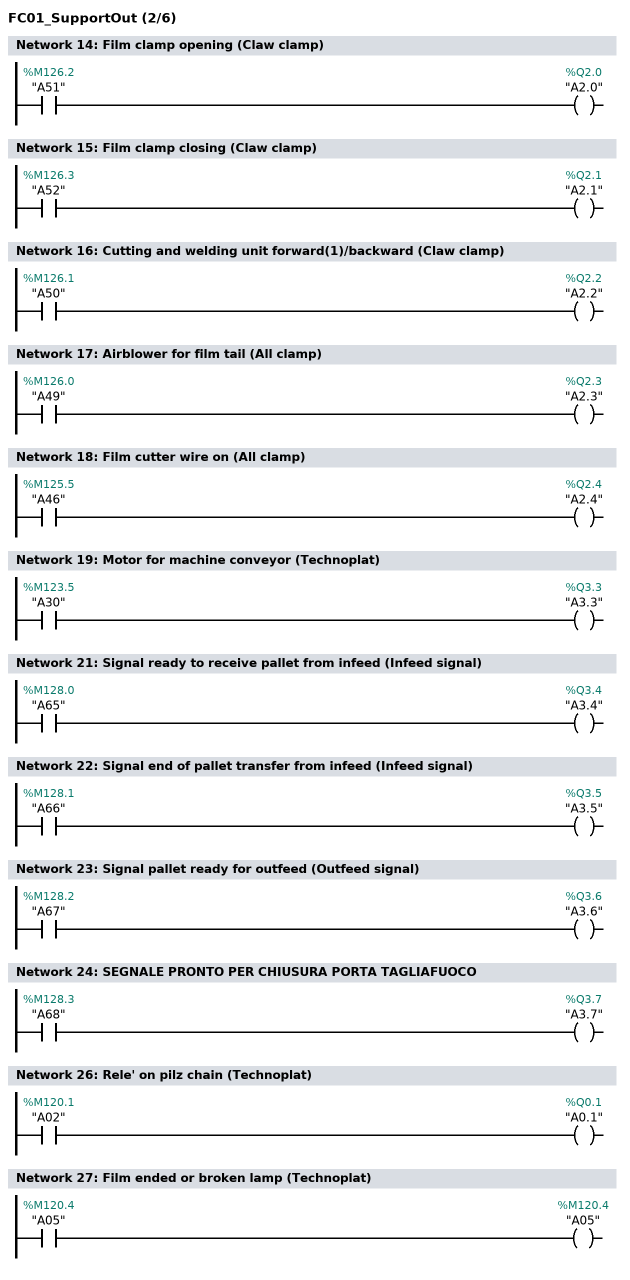
   RUNG wire#powerrail
      Contact( "A51" )
      Coil( "A2.0" )
   END_RUNG
   // the same network as SCL:
   "A2.0" := "A51";
END_REGION

REGION Network 15: Film clamp closing (Claw clamp)
   RUNG wire#powerrail
      Contact( "A52" )
      Coil( "A2.1" )
   END_RUNG
   // the same network as SCL:
   "A2.1" := "A52";
END_REGION

REGION Network 16: Cutting and welding unit forward(1)/backward (Claw clamp)
   RUNG wire#powerrail
      Contact( "A50" )
      Coil( "A2.2" )
   END_RUNG
   // the same network as SCL:
   "A2.2" := "A50";
END_REGION

REGION Network 17: Airblower for film tail (All clamp)
   RUNG wire#powerrail
      Contact( "A49" )
      Coil( "A2.3" )
   END_RUNG
   // the same network as SCL:
   "A2.3" := "A49";
END_REGION

REGION Network 18: Film cutter wire on (All clamp)
   RUNG wire#powerrail
      Contact( "A46" )
      Coil( "A2.4" )
   END_RUNG
   // the same network as SCL:
   "A2.4" := "A46";
END_REGION

REGION Network 19: Motor for machine conveyor (Technoplat)
   RUNG wire#powerrail
      Contact( "A30" )
      Coil( "A3.3" )
   END_RUNG
   // the same network as SCL:
   "A3.3" := "A30";
END_REGION

REGION Network 20: EXCHANGE SIGNALS
END_REGION

REGION Network 21: Signal ready to receive pallet from infeed (Infeed signal)
   RUNG wire#powerrail
      Contact( "A65" )
      Coil( "A3.4" )
   END_RUNG
   // the same network as SCL:
   "A3.4" := "A65";
END_REGION

REGION Network 22: Signal end of pallet transfer from infeed (Infeed signal)
   RUNG wire#powerrail
      Contact( "A66" )
      Coil( "A3.5" )
   END_RUNG
   // the same network as SCL:
   "A3.5" := "A66";
END_REGION

REGION Network 23: Signal pallet ready for outfeed (Outfeed signal)
   RUNG wire#powerrail
      Contact( "A67" )
      Coil( "A3.6" )
   END_RUNG
   // the same network as SCL:
   "A3.6" := "A67";
END_REGION

REGION Network 24: SEGNALE PRONTO PER CHIUSURA PORTA TAGLIAFUOCO
   RUNG wire#powerrail
      Contact( "A68" )
      Coil( "A3.7" )
   END_RUNG
   // the same network as SCL:
   "A3.7" := "A68";
END_REGION

REGION Network 25: ACCESSORIES
END_REGION

REGION Network 26: Rele' on pilz chain (Technoplat)
   RUNG wire#powerrail
      Contact( "A02" )
      Coil( "A0.1" )
   END_RUNG
   // the same network as SCL:
   "A0.1" := "A02";
END_REGION

REGION Network 27: Film ended or broken lamp (Technoplat)
   RUNG wire#powerrail
      Contact( "A05" )
      Coil( "A05" )
   END_RUNG
   // the same network as SCL:
   "A05" := "A05";
END_REGION

REGION Network 28: ***DOOR***
END_REGION

REGION Network 29: Request to open door (Technoplat)
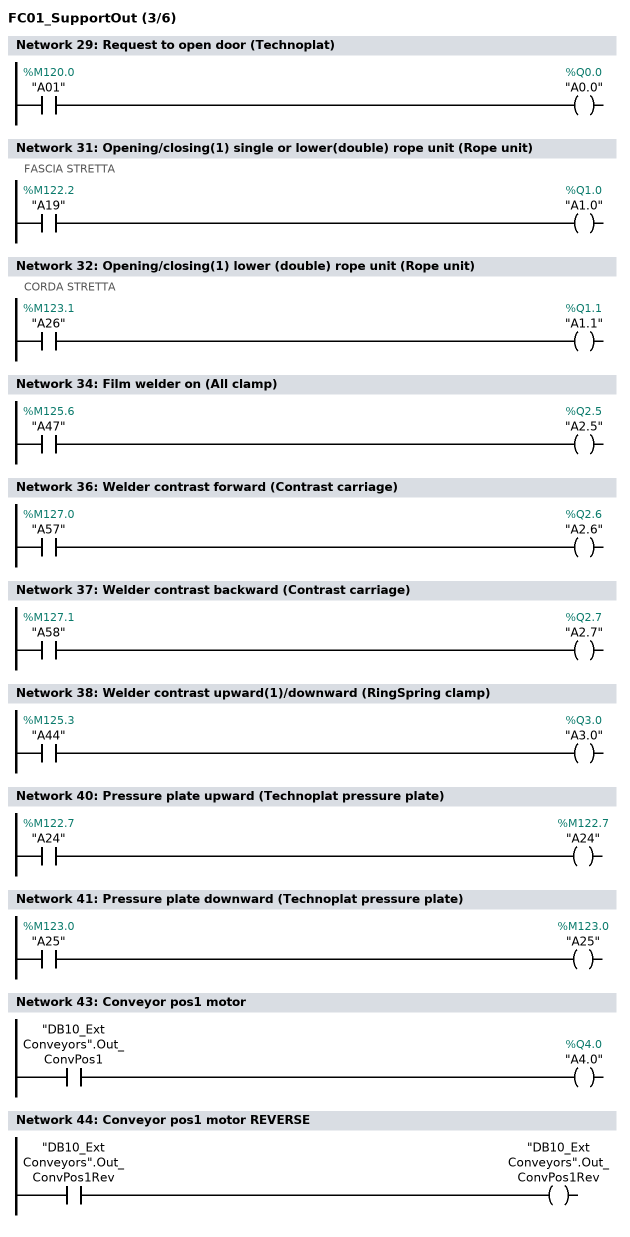
   RUNG wire#powerrail
      Contact( "A01" )
      Coil( "A0.0" )
   END_RUNG
   // the same network as SCL:
   "A0.0" := "A01";
END_REGION

REGION Network 30: ***BAND/ROPE***
END_REGION

REGION Network 31: Opening/closing(1) single or lower(double) rope unit (Rope unit)
   // FASCIA STRETTA
   RUNG wire#powerrail
      Contact( "A19" )
      Coil( "A1.0" )
   END_RUNG
   // the same network as SCL:
   "A1.0" := "A19";
END_REGION

REGION Network 32: Opening/closing(1) lower (double) rope unit (Rope unit)
   // CORDA STRETTA
   RUNG wire#powerrail
      Contact( "A26" )
      Coil( "A1.1" )
   END_RUNG
   // the same network as SCL:
   "A1.1" := "A26";
END_REGION

REGION Network 33: ***WELDER***
END_REGION

REGION Network 34: Film welder on (All clamp)
   RUNG wire#powerrail
      Contact( "A47" )
      Coil( "A2.5" )
   END_RUNG
   // the same network as SCL:
   "A2.5" := "A47";
END_REGION

REGION Network 35: ***CONTRAST***
END_REGION

REGION Network 36: Welder contrast forward (Contrast carriage)
   RUNG wire#powerrail
      Contact( "A57" )
      Coil( "A2.6" )
   END_RUNG
   // the same network as SCL:
   "A2.6" := "A57";
END_REGION

REGION Network 37: Welder contrast backward (Contrast carriage)
   RUNG wire#powerrail
      Contact( "A58" )
      Coil( "A2.7" )
   END_RUNG
   // the same network as SCL:
   "A2.7" := "A58";
END_REGION

REGION Network 38: Welder contrast upward(1)/downward (RingSpring clamp)
   RUNG wire#powerrail
      Contact( "A44" )
      Coil( "A3.0" )
   END_RUNG
   // the same network as SCL:
   "A3.0" := "A44";
END_REGION

REGION Network 39: ***PRESSURE***
END_REGION

REGION Network 40: Pressure plate upward (Technoplat pressure plate)
   RUNG wire#powerrail
      Contact( "A24" )
      Coil( "A24" )
   END_RUNG
   // the same network as SCL:
   "A24" := "A24";
END_REGION

REGION Network 41: Pressure plate downward (Technoplat pressure plate)
   RUNG wire#powerrail
      Contact( "A25" )
      Coil( "A25" )
   END_RUNG
   // the same network as SCL:
   "A25" := "A25";
END_REGION

REGION Network 42: ***CONVEYORS***
END_REGION

REGION Network 43: Conveyor pos1 motor
   RUNG wire#powerrail
      Contact( "DB10_ExtConveyors".Out_ConvPos1 )
      Coil( "A4.0" )
   END_RUNG
   // the same network as SCL:
   "A4.0" := "DB10_ExtConveyors".Out_ConvPos1;
END_REGION

REGION Network 44: Conveyor pos1 motor REVERSE
   RUNG wire#powerrail
      Contact( "DB10_ExtConveyors".Out_ConvPos1Rev )
      Coil( "DB10_ExtConveyors".Out_ConvPos1Rev )
   END_RUNG
   // the same network as SCL:
   "DB10_ExtConveyors".Out_ConvPos1Rev := "DB10_ExtConveyors".Out_ConvPos1Rev;
END_REGION

REGION Network 45: Conveyor pos1 motor speed selection X2
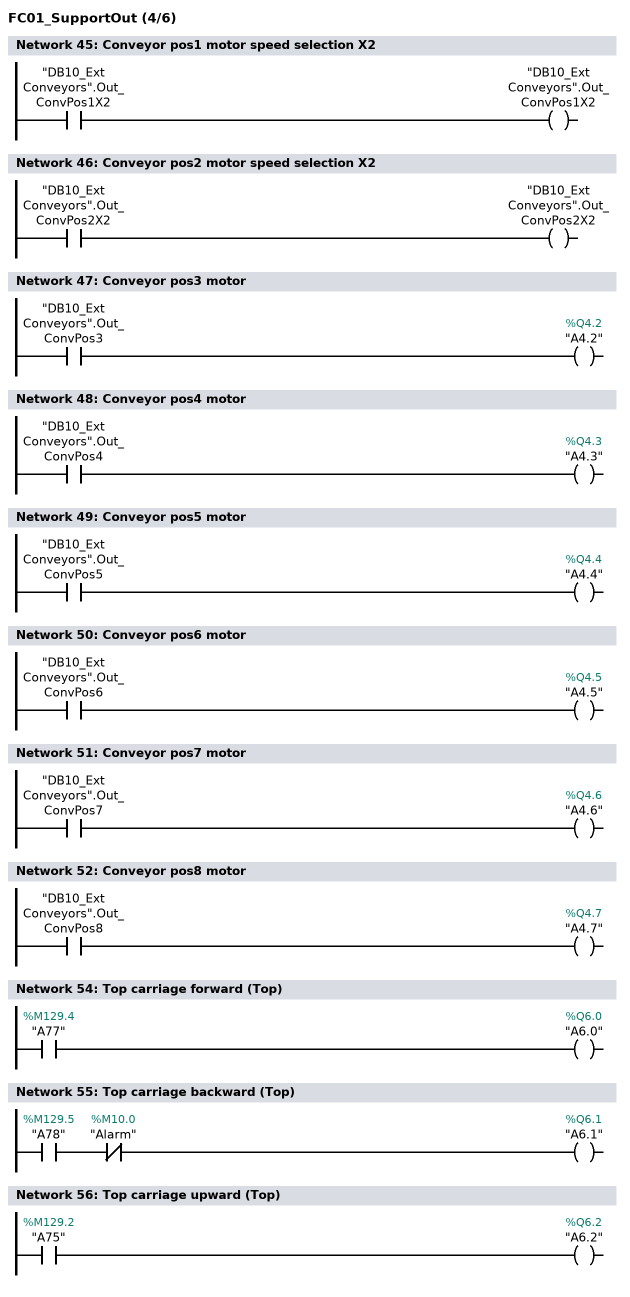
   RUNG wire#powerrail
      Contact( "DB10_ExtConveyors".Out_ConvPos1X2 )
      Coil( "DB10_ExtConveyors".Out_ConvPos1X2 )
   END_RUNG
   // the same network as SCL:
   "DB10_ExtConveyors".Out_ConvPos1X2 := "DB10_ExtConveyors".Out_ConvPos1X2;
END_REGION

REGION Network 46: Conveyor pos2 motor speed selection X2
   RUNG wire#powerrail
      Contact( "DB10_ExtConveyors".Out_ConvPos2X2 )
      Coil( "DB10_ExtConveyors".Out_ConvPos2X2 )
   END_RUNG
   // the same network as SCL:
   "DB10_ExtConveyors".Out_ConvPos2X2 := "DB10_ExtConveyors".Out_ConvPos2X2;
END_REGION

REGION Network 47: Conveyor pos3 motor
   RUNG wire#powerrail
      Contact( "DB10_ExtConveyors".Out_ConvPos3 )
      Coil( "A4.2" )
   END_RUNG
   // the same network as SCL:
   "A4.2" := "DB10_ExtConveyors".Out_ConvPos3;
END_REGION

REGION Network 48: Conveyor pos4 motor
   RUNG wire#powerrail
      Contact( "DB10_ExtConveyors".Out_ConvPos4 )
      Coil( "A4.3" )
   END_RUNG
   // the same network as SCL:
   "A4.3" := "DB10_ExtConveyors".Out_ConvPos4;
END_REGION

REGION Network 49: Conveyor pos5 motor
   RUNG wire#powerrail
      Contact( "DB10_ExtConveyors".Out_ConvPos5 )
      Coil( "A4.4" )
   END_RUNG
   // the same network as SCL:
   "A4.4" := "DB10_ExtConveyors".Out_ConvPos5;
END_REGION

REGION Network 50: Conveyor pos6 motor
   RUNG wire#powerrail
      Contact( "DB10_ExtConveyors".Out_ConvPos6 )
      Coil( "A4.5" )
   END_RUNG
   // the same network as SCL:
   "A4.5" := "DB10_ExtConveyors".Out_ConvPos6;
END_REGION

REGION Network 51: Conveyor pos7 motor
   RUNG wire#powerrail
      Contact( "DB10_ExtConveyors".Out_ConvPos7 )
      Coil( "A4.6" )
   END_RUNG
   // the same network as SCL:
   "A4.6" := "DB10_ExtConveyors".Out_ConvPos7;
END_REGION

REGION Network 52: Conveyor pos8 motor
   RUNG wire#powerrail
      Contact( "DB10_ExtConveyors".Out_ConvPos8 )
      Coil( "A4.7" )
   END_RUNG
   // the same network as SCL:
   "A4.7" := "DB10_ExtConveyors".Out_ConvPos8;
END_REGION

REGION Network 53: ***TOP***
END_REGION

REGION Network 54: Top carriage forward (Top)
   RUNG wire#powerrail
      Contact( "A77" )
      Coil( "A6.0" )
   END_RUNG
   // the same network as SCL:
   "A6.0" := "A77";
END_REGION

REGION Network 55: Top carriage backward (Top)
   RUNG wire#powerrail
      Contact( "A78" )
      I_Contact( "Alarm" )
      Coil( "A6.1" )
   END_RUNG
   // the same network as SCL:
   "A6.1" := "A78" AND NOT "Alarm";
END_REGION

REGION Network 56: Top carriage upward (Top)
   RUNG wire#powerrail
      Contact( "A75" )
      Coil( "A6.2" )
   END_RUNG
   // the same network as SCL:
   "A6.2" := "A75";
END_REGION

REGION Network 57: Top carriage downward (Top)
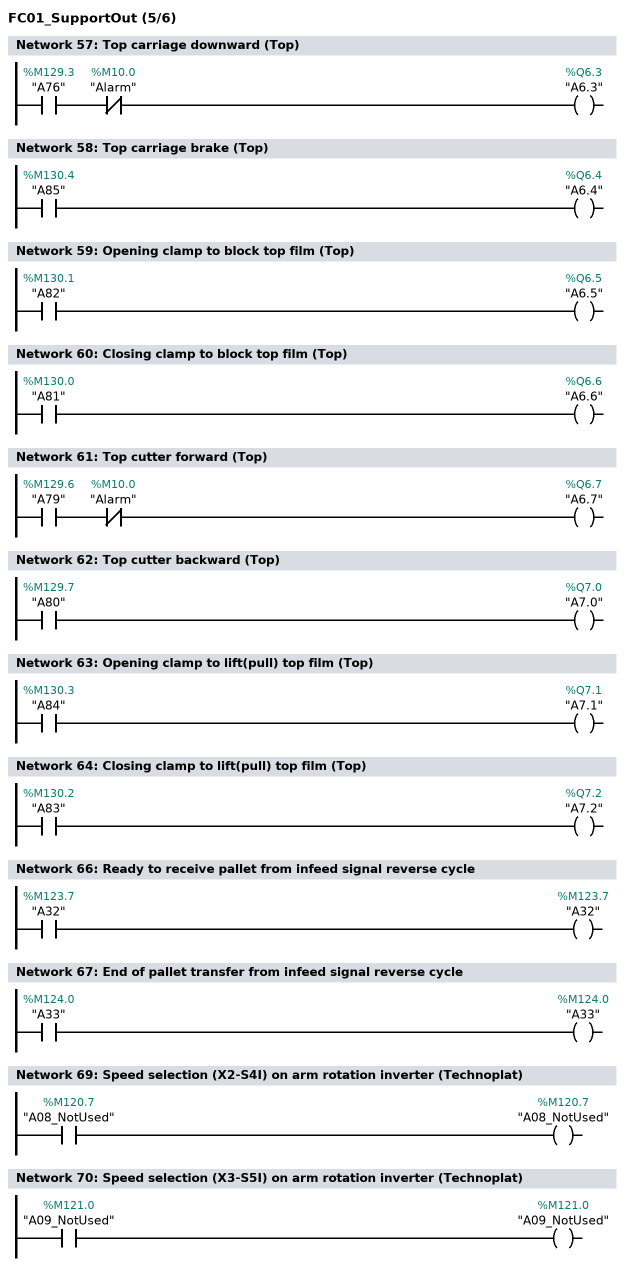
   RUNG wire#powerrail
      Contact( "A76" )
      I_Contact( "Alarm" )
      Coil( "A6.3" )
   END_RUNG
   // the same network as SCL:
   "A6.3" := "A76" AND NOT "Alarm";
END_REGION

REGION Network 58: Top carriage brake (Top)
   RUNG wire#powerrail
      Contact( "A85" )
      Coil( "A6.4" )
   END_RUNG
   // the same network as SCL:
   "A6.4" := "A85";
END_REGION

REGION Network 59: Opening clamp to block top film (Top)
   RUNG wire#powerrail
      Contact( "A82" )
      Coil( "A6.5" )
   END_RUNG
   // the same network as SCL:
   "A6.5" := "A82";
END_REGION

REGION Network 60: Closing clamp to block top film (Top)
   RUNG wire#powerrail
      Contact( "A81" )
      Coil( "A6.6" )
   END_RUNG
   // the same network as SCL:
   "A6.6" := "A81";
END_REGION

REGION Network 61: Top cutter forward (Top)
   RUNG wire#powerrail
      Contact( "A79" )
      I_Contact( "Alarm" )
      Coil( "A6.7" )
   END_RUNG
   // the same network as SCL:
   "A6.7" := "A79" AND NOT "Alarm";
END_REGION

REGION Network 62: Top cutter backward (Top)
   RUNG wire#powerrail
      Contact( "A80" )
      Coil( "A7.0" )
   END_RUNG
   // the same network as SCL:
   "A7.0" := "A80";
END_REGION

REGION Network 63: Opening clamp to lift(pull) top film (Top)
   RUNG wire#powerrail
      Contact( "A84" )
      Coil( "A7.1" )
   END_RUNG
   // the same network as SCL:
   "A7.1" := "A84";
END_REGION

REGION Network 64: Closing clamp to lift(pull) top film (Top)
   RUNG wire#powerrail
      Contact( "A83" )
      Coil( "A7.2" )
   END_RUNG
   // the same network as SCL:
   "A7.2" := "A83";
END_REGION

REGION Network 65: OTHER
END_REGION

REGION Network 66: Ready to receive pallet from infeed signal reverse cycle
   RUNG wire#powerrail
      Contact( "A32" )
      Coil( "A32" )
   END_RUNG
   // the same network as SCL:
   "A32" := "A32";
END_REGION

REGION Network 67: End of pallet transfer from infeed signal reverse cycle
   RUNG wire#powerrail
      Contact( "A33" )
      Coil( "A33" )
   END_RUNG
   // the same network as SCL:
   "A33" := "A33";
END_REGION

REGION Network 68: OLD (NOT USED)
END_REGION

REGION Network 69: Speed selection (X2-S4I) on arm rotation inverter (Technoplat)
   RUNG wire#powerrail
      Contact( "A08_NotUsed" )
      Coil( "A08_NotUsed" )
   END_RUNG
   // the same network as SCL:
   "A08_NotUsed" := "A08_NotUsed";
END_REGION

REGION Network 70: Speed selection (X3-S5I) on arm rotation inverter (Technoplat)
   RUNG wire#powerrail
      Contact( "A09_NotUsed" )
      Coil( "A09_NotUsed" )
   END_RUNG
   // the same network as SCL:
   "A09_NotUsed" := "A09_NotUsed";
END_REGION

REGION Network 71: Pallet lifter upward(1)/downard (Lifter)
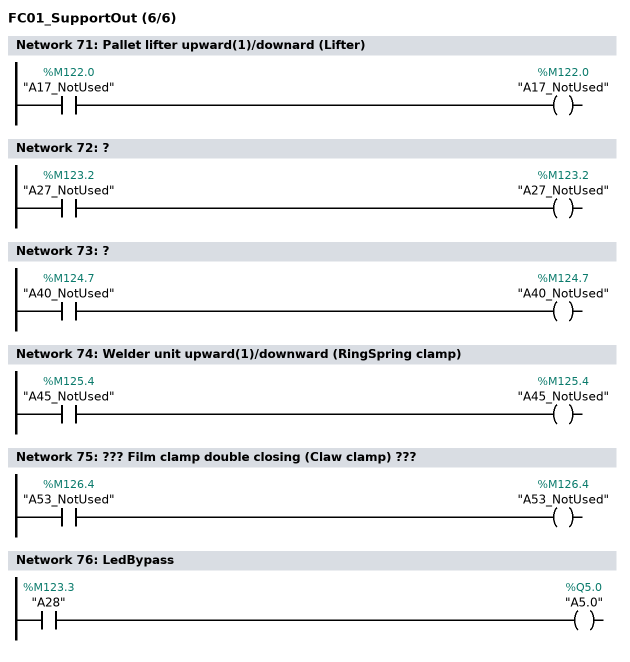
   RUNG wire#powerrail
      Contact( "A17_NotUsed" )
      Coil( "A17_NotUsed" )
   END_RUNG
   // the same network as SCL:
   "A17_NotUsed" := "A17_NotUsed";
END_REGION

REGION Network 72: ?
   RUNG wire#powerrail
      Contact( "A27_NotUsed" )
      Coil( "A27_NotUsed" )
   END_RUNG
   // the same network as SCL:
   "A27_NotUsed" := "A27_NotUsed";
END_REGION

REGION Network 73: ?
   RUNG wire#powerrail
      Contact( "A40_NotUsed" )
      Coil( "A40_NotUsed" )
   END_RUNG
   // the same network as SCL:
   "A40_NotUsed" := "A40_NotUsed";
END_REGION

REGION Network 74: Welder unit upward(1)/downward (RingSpring clamp)
   RUNG wire#powerrail
      Contact( "A45_NotUsed" )
      Coil( "A45_NotUsed" )
   END_RUNG
   // the same network as SCL:
   "A45_NotUsed" := "A45_NotUsed";
END_REGION

REGION Network 75: ??? Film clamp double closing (Claw clamp) ???
   RUNG wire#powerrail
      Contact( "A53_NotUsed" )
      Coil( "A53_NotUsed" )
   END_RUNG
   // the same network as SCL:
   "A53_NotUsed" := "A53_NotUsed";
END_REGION

REGION Network 76: LedBypass
   RUNG wire#powerrail
      Contact( "A28" )
      Coil( "A5.0" )
   END_RUNG
   // the same network as SCL:
   "A5.0" := "A28";
END_REGION
END_FUNCTION

FUNCTION_BLOCK "Centrador_Paletes"   // FB2, LAD
TITLE = CONTROLO DE CENTRADOR DE PALETES
{ S7_Optimized_Access := 'TRUE' }
VERSION : 0.1
// stored: AutoNumber true, IsIECCheckEnabled false, IsRetainMemResEnabled false, MemoryReserve 100, SetENOAutomatically false, UDAEnableTagReadback false
   VAR_INPUT
      Centrador_Aberto_1 : Bool;
      Centrador_Aberto_2 : Bool;
      Detetor_Palete : Bool;
      Palete_Centrada_1 : Bool;
      Palete_Centrada_2 : Bool;
   END_VAR
   VAR_OUTPUT
      "ETAPA 1 (INICIO)" : Bool := true;
      "ETAPA 2" : Bool;
      "ETAPA 3" : Bool;
      "ETAPA 4" : Bool;
      Motor_Tapete_Centrador : Bool;
      Motor_Centrador_Sentido_Direto : Bool;
      Motor_Centrador_Sentido_Inverso : Bool;
   END_VAR
   VAR_TEMP   // added for the SCL form of the ladder/FBD networks
      _w1 : Bool;
   END_VAR
BEGIN

REGION Network 1: ETAPA 2 - Arranque de tapete do centrador
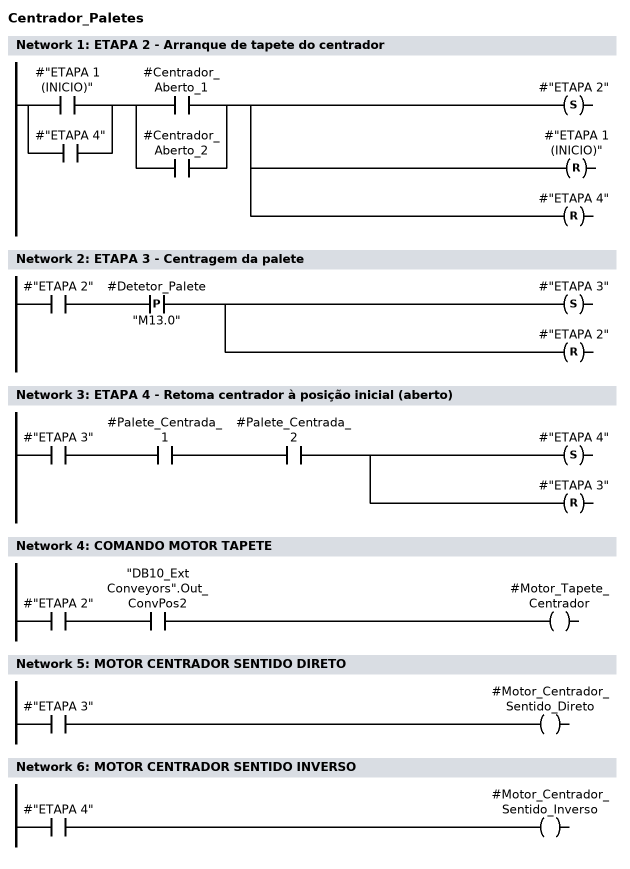
   RUNG wire#powerrail
      Contact( #"ETAPA 1 (INICIO)" )
      wire#w1
      Contact( #Centrador_Aberto_1 )
      wire#w2
      S_Coil( #"ETAPA 2" )
   END_RUNG
   RUNG wire#powerrail
      Contact( #"ETAPA 4" )
   END_RUNG wire#w1
   RUNG wire#w1
      Contact( #Centrador_Aberto_2 )
   END_RUNG wire#w2
   RUNG wire#w2
      R_Coil( #"ETAPA 1 (INICIO)" )
   END_RUNG
   RUNG wire#w2
      R_Coil( #"ETAPA 4" )
   END_RUNG
   // the same network as SCL:
   IF (#"ETAPA 1 (INICIO)" OR #"ETAPA 4") AND (#Centrador_Aberto_1 OR #Centrador_Aberto_2) THEN
       #"ETAPA 2" := TRUE;
   END_IF;
   #_w1 := (#"ETAPA 1 (INICIO)" OR #"ETAPA 4") AND (#Centrador_Aberto_1 OR #Centrador_Aberto_2);
   IF #_w1 THEN
       #"ETAPA 1 (INICIO)" := FALSE;
       #"ETAPA 4" := FALSE;
   END_IF;
END_REGION

REGION Network 2: ETAPA 3 - Centragem da palete
   RUNG wire#powerrail
      Contact( #"ETAPA 2" )
      P_Contact(operand := #Detetor_Palete, bit := "M13.0")
      wire#w1
      S_Coil( #"ETAPA 3" )
   END_RUNG
   RUNG wire#w1
      R_Coil( #"ETAPA 2" )
   END_RUNG
   // the same network as SCL:
   #_w1 := #"ETAPA 2" AND #Detetor_Palete AND NOT "M13.0";   // rising edge of #Detetor_Palete
   "M13.0" := #Detetor_Palete;
   IF #_w1 THEN
       #"ETAPA 3" := TRUE;
       #"ETAPA 2" := FALSE;
   END_IF;
END_REGION

REGION Network 3: ETAPA 4 - Retoma centrador à posição inicial (aberto)
   RUNG wire#powerrail
      Contact( #"ETAPA 3" )
      Contact( #Palete_Centrada_1 )
      Contact( #Palete_Centrada_2 )
      wire#w1
      S_Coil( #"ETAPA 4" )
   END_RUNG
   RUNG wire#w1
      R_Coil( #"ETAPA 3" )
   END_RUNG
   // the same network as SCL:
   IF #"ETAPA 3" AND #Palete_Centrada_1 AND #Palete_Centrada_2 THEN
       #"ETAPA 4" := TRUE;
       #"ETAPA 3" := FALSE;
   END_IF;
END_REGION

REGION Network 4: COMANDO MOTOR TAPETE
   RUNG wire#powerrail
      Contact( #"ETAPA 2" )
      Contact( "DB10_ExtConveyors".Out_ConvPos2 )
      Coil( #Motor_Tapete_Centrador )
   END_RUNG
   // the same network as SCL:
   #Motor_Tapete_Centrador := #"ETAPA 2" AND "DB10_ExtConveyors".Out_ConvPos2;
END_REGION

REGION Network 5: MOTOR CENTRADOR SENTIDO DIRETO
   RUNG wire#powerrail
      Contact( #"ETAPA 3" )
      Coil( #Motor_Centrador_Sentido_Direto )
   END_RUNG
   // the same network as SCL:
   #Motor_Centrador_Sentido_Direto := #"ETAPA 3";
END_REGION

REGION Network 6: MOTOR CENTRADOR SENTIDO INVERSO
   RUNG wire#powerrail
      Contact( #"ETAPA 4" )
      Coil( #Motor_Centrador_Sentido_Inverso )
   END_RUNG
   // the same network as SCL:
   #Motor_Centrador_Sentido_Inverso := #"ETAPA 4";
END_REGION
END_FUNCTION_BLOCK

ORGANIZATION_BLOCK "Cyclic interrupt"   // OB30, LAD, CyclicInterrupt
TITLE = Rampa tiro
{ S7_Optimized_Access := 'TRUE' }
VERSION : 0.1
// Rampa per raggiungere tiro obiettivo e zero (0-20@100ms;20-100@20ms->3600ms)
// stored: AutoNumber true, IsIECCheckEnabled false, SetENOAutomatically false
   VAR_INPUT
      Initial_Call : Bool;   // Initial call of this OB
      Event_Count : Int;   // Events discarded
   END_VAR
   VAR_TEMP
      TempDint : DInt;
      TempDint_2 : DInt;
      TempInt : Int;
   END_VAR
   VAR_TEMP   // added for the SCL form of the ladder/FBD networks
      _w1 : Bool;
      _w2 : Bool;
   END_VAR
BEGIN

REGION Network 1: Impulso ogni 20ms (OB30)
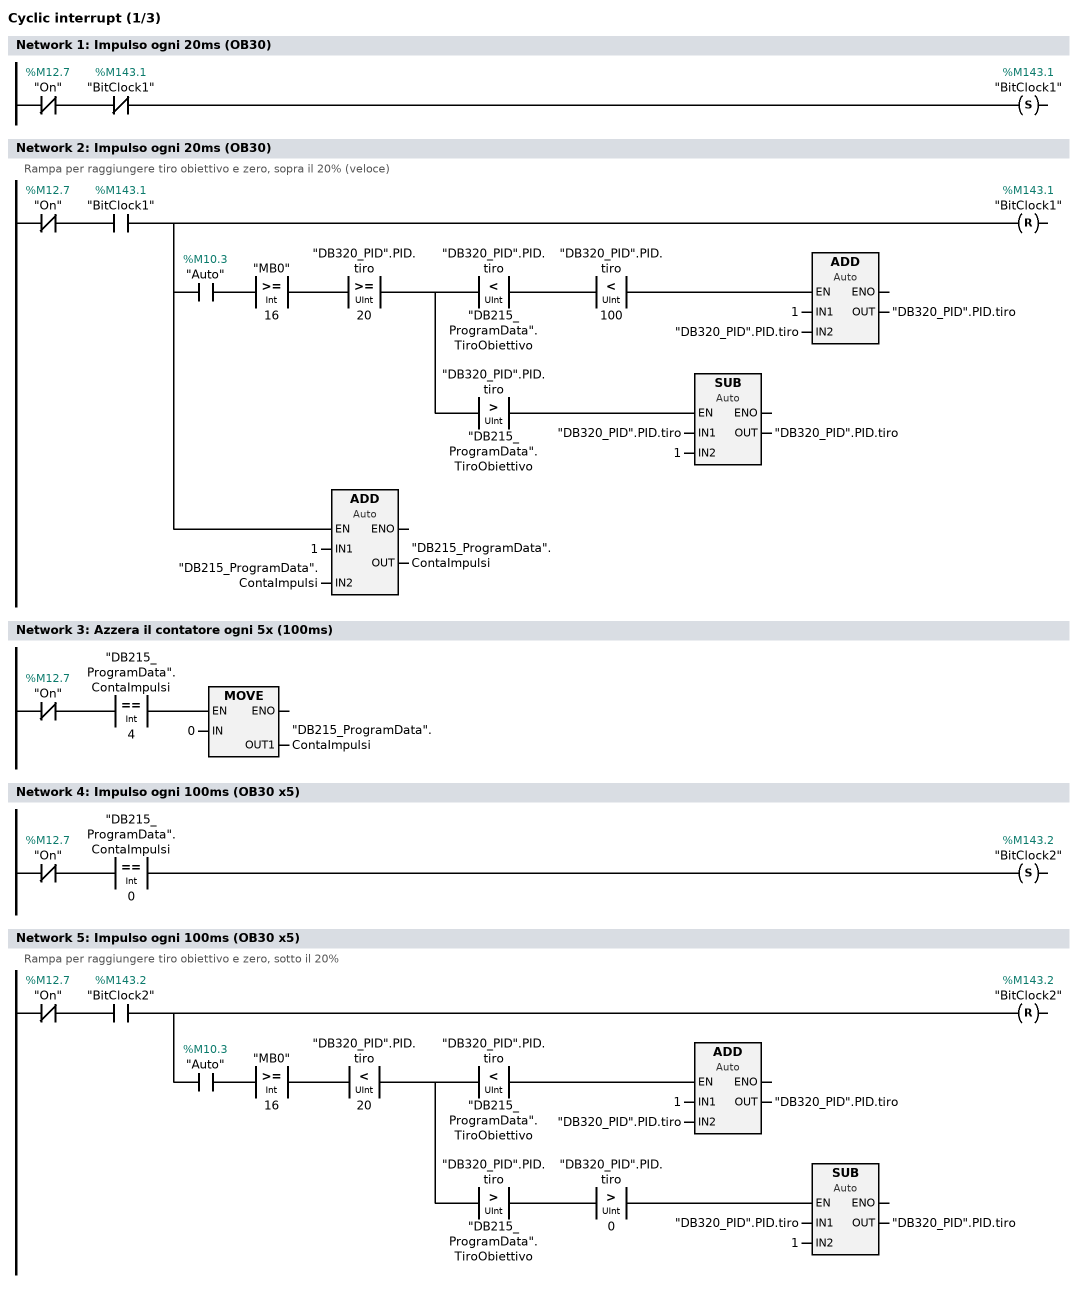
   RUNG wire#powerrail
      I_Contact( "On" )
      I_Contact( "BitClock1" )
      S_Coil( "BitClock1" )
   END_RUNG
   // the same network as SCL:
   IF NOT "On" AND NOT "BitClock1" THEN "BitClock1" := TRUE; END_IF;
END_REGION

REGION Network 2: Impulso ogni 20ms (OB30)
   // Rampa per raggiungere tiro obiettivo e zero, sopra il 20% (veloce)
   RUNG wire#powerrail
      I_Contact( "On" )
      Contact( "BitClock1" )
      wire#w1
      R_Coil( "BitClock1" )
   END_RUNG
   RUNG wire#w1
      Contact( "Auto" )
      { S7_Templates := "SrcType := Int" } GE_Contact(in1 := "MB0", in2 := 16)
      { S7_Templates := "SrcType := UInt" } GE_Contact(in1 := "DB320_PID".PID.tiro, in2 := 20)
      wire#w2
      { S7_Templates := "SrcType := UInt" } LT_Contact(in1 := "DB320_PID".PID.tiro, in2 := "DB215_ProgramData".TiroObiettivo)
      { S7_Templates := "SrcType := UInt" } LT_Contact(in1 := "DB320_PID".PID.tiro, in2 := 100)
      Add(in1 := 1, in2 := "DB320_PID".PID.tiro, out => "DB320_PID".PID.tiro)
   END_RUNG
   RUNG wire#w2
      { S7_Templates := "SrcType := UInt" } GT_Contact(in1 := "DB320_PID".PID.tiro, in2 := "DB215_ProgramData".TiroObiettivo)
      Sub(in1 := "DB320_PID".PID.tiro, in2 := 1, out => "DB320_PID".PID.tiro)
   END_RUNG
   RUNG wire#w1
      Add(in1 := 1, in2 := "DB215_ProgramData".ContaImpulsi, out => "DB215_ProgramData".ContaImpulsi)
   END_RUNG
   // the same network as SCL:
   #_w1 := NOT "On" AND "BitClock1";
   IF #_w1 THEN "BitClock1" := FALSE; END_IF;
   #_w2 := #_w1 AND "Auto" AND ("MB0" >= 16) AND ("DB320_PID".PID.tiro >= 20);
   IF #_w2 AND ("DB320_PID".PID.tiro < "DB215_ProgramData".TiroObiettivo) AND ("DB320_PID".PID.tiro < 100) THEN
       "DB320_PID".PID.tiro := 1 + "DB320_PID".PID.tiro;
   END_IF;
   IF #_w2 AND ("DB320_PID".PID.tiro > "DB215_ProgramData".TiroObiettivo) THEN
       "DB320_PID".PID.tiro := "DB320_PID".PID.tiro - 1;
   END_IF;
   IF #_w1 THEN "DB215_ProgramData".ContaImpulsi := 1 + "DB215_ProgramData".ContaImpulsi; END_IF;
END_REGION

REGION Network 3: Azzera il contatore ogni 5x (100ms)
   RUNG wire#powerrail
      I_Contact( "On" )
      { S7_Templates := "SrcType := Int" } EQ_Contact(in1 := "DB215_ProgramData".ContaImpulsi, in2 := 4)
      Move(in := 0, out1 => "DB215_ProgramData".ContaImpulsi)
   END_RUNG
   // the same network as SCL:
   IF NOT "On" AND ("DB215_ProgramData".ContaImpulsi = 4) THEN "DB215_ProgramData".ContaImpulsi := 0; END_IF;
END_REGION

REGION Network 4: Impulso ogni 100ms (OB30 x5)
   RUNG wire#powerrail
      I_Contact( "On" )
      { S7_Templates := "SrcType := Int" } EQ_Contact(in1 := "DB215_ProgramData".ContaImpulsi, in2 := 0)
      S_Coil( "BitClock2" )
   END_RUNG
   // the same network as SCL:
   IF NOT "On" AND ("DB215_ProgramData".ContaImpulsi = 0) THEN "BitClock2" := TRUE; END_IF;
END_REGION

REGION Network 5: Impulso ogni 100ms (OB30 x5)
   // Rampa per raggiungere tiro obiettivo e zero, sotto il 20%
   RUNG wire#powerrail
      I_Contact( "On" )
      Contact( "BitClock2" )
      wire#w1
      R_Coil( "BitClock2" )
   END_RUNG
   RUNG wire#w1
      Contact( "Auto" )
      { S7_Templates := "SrcType := Int" } GE_Contact(in1 := "MB0", in2 := 16)
      { S7_Templates := "SrcType := UInt" } LT_Contact(in1 := "DB320_PID".PID.tiro, in2 := 20)
      wire#w2
      { S7_Templates := "SrcType := UInt" } LT_Contact(in1 := "DB320_PID".PID.tiro, in2 := "DB215_ProgramData".TiroObiettivo)
      Add(in1 := 1, in2 := "DB320_PID".PID.tiro, out => "DB320_PID".PID.tiro)
   END_RUNG
   RUNG wire#w2
      { S7_Templates := "SrcType := UInt" } GT_Contact(in1 := "DB320_PID".PID.tiro, in2 := "DB215_ProgramData".TiroObiettivo)
      { S7_Templates := "SrcType := UInt" } GT_Contact(in1 := "DB320_PID".PID.tiro, in2 := 0)
      Sub(in1 := "DB320_PID".PID.tiro, in2 := 1, out => "DB320_PID".PID.tiro)
   END_RUNG
   // the same network as SCL:
   #_w1 := NOT "On" AND "BitClock2";
   IF #_w1 THEN "BitClock2" := FALSE; END_IF;
   #_w2 := #_w1 AND "Auto" AND ("MB0" >= 16) AND ("DB320_PID".PID.tiro < 20);
   IF #_w2 AND ("DB320_PID".PID.tiro < "DB215_ProgramData".TiroObiettivo) THEN
       "DB320_PID".PID.tiro := 1 + "DB320_PID".PID.tiro;
   END_IF;
   IF #_w2 AND ("DB320_PID".PID.tiro > "DB215_ProgramData".TiroObiettivo) AND ("DB320_PID".PID.tiro > 0) THEN
       "DB320_PID".PID.tiro := "DB320_PID".PID.tiro - 1;
   END_IF;
END_REGION

REGION Network 7: Arm rotation and top carriage speed change for DAC M20
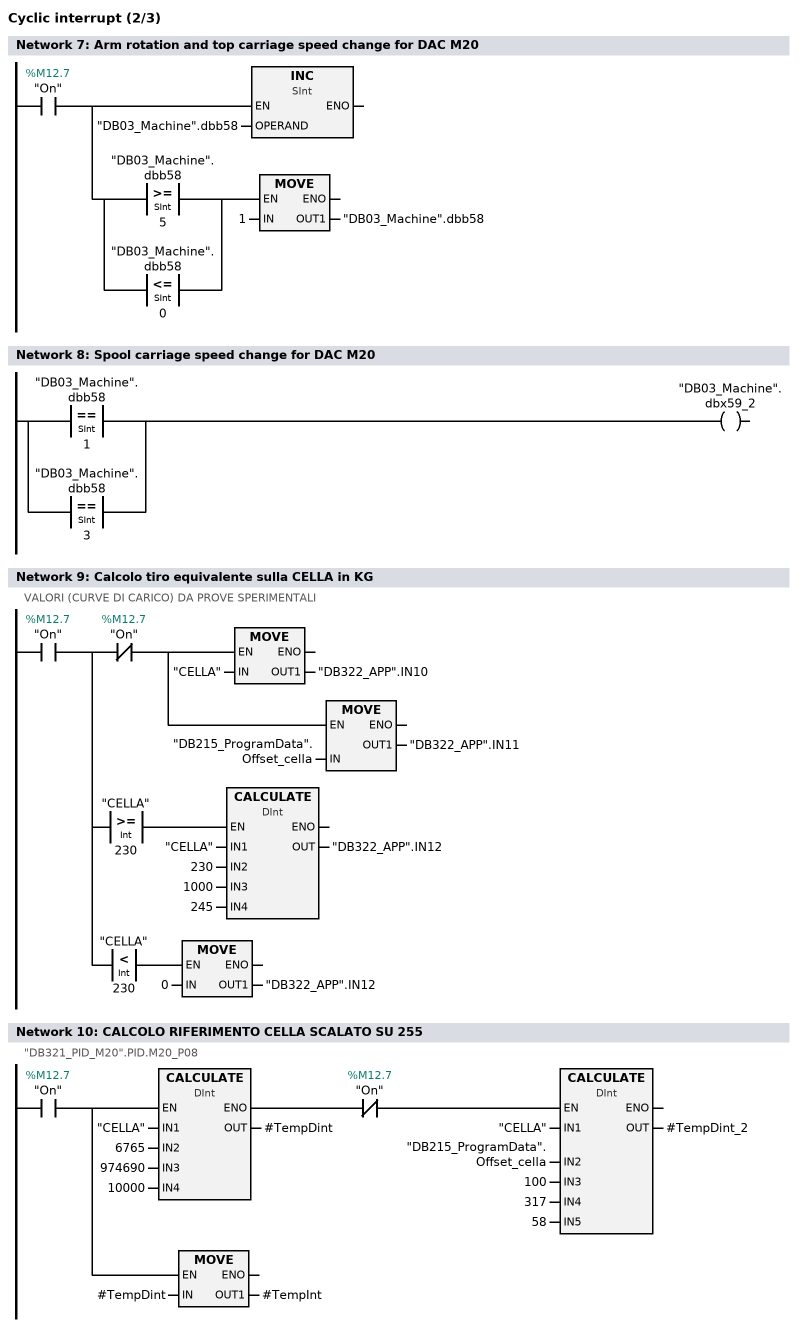
   RUNG wire#powerrail
      Contact( "On" )
      wire#w1
      { S7_Templates := "DestType := SInt"; S7_GenerateENO := "TRUE" } Inc( "DB03_Machine".dbb58 )
   END_RUNG
   RUNG wire#w1
      { S7_Templates := "SrcType := SInt" } GE_Contact(in1 := "DB03_Machine".dbb58, in2 := 5)
      wire#w2
      { S7_GenerateENO := "TRUE" } Move(in := 1, out1 => "DB03_Machine".dbb58)
   END_RUNG
   RUNG wire#w1
      { S7_Templates := "SrcType := SInt" } LE_Contact(in1 := "DB03_Machine".dbb58, in2 := 0)
   END_RUNG wire#w2
   // the same network as SCL:
   IF "On" THEN "DB03_Machine".dbb58 := "DB03_Machine".dbb58 + 1; END_IF;
   IF "On" AND (("DB03_Machine".dbb58 >= 5) OR ("DB03_Machine".dbb58 <= 0)) THEN
       "DB03_Machine".dbb58 := 1;
   END_IF;
END_REGION

REGION Network 8: Spool carriage speed change for DAC M20
   RUNG wire#powerrail
      { S7_Templates := "SrcType := SInt" } EQ_Contact(in1 := "DB03_Machine".dbb58, in2 := 1)
      wire#w1
      Coil( "DB03_Machine".dbx59_2 )
   END_RUNG
   RUNG wire#powerrail
      { S7_Templates := "SrcType := SInt" } EQ_Contact(in1 := "DB03_Machine".dbb58, in2 := 3)
   END_RUNG wire#w1
   // the same network as SCL:
   "DB03_Machine".dbx59_2 := ("DB03_Machine".dbb58 = 1) OR ("DB03_Machine".dbb58 = 3);
END_REGION

REGION Network 9: Calcolo tiro equivalente sulla CELLA in KG
   // VALORI (CURVE DI CARICO) DA PROVE SPERIMENTALI
   RUNG wire#powerrail
      Contact( "On" )
      wire#w1
      I_Contact( "On" )
      wire#w2
      Move(in := "CELLA", out1 => "DB322_APP".IN10)
   END_RUNG
   RUNG wire#w2
      Move(in := "DB215_ProgramData".Offset_cella, out1 => "DB322_APP".IN11)
   END_RUNG
   RUNG wire#w1
      { S7_Templates := "SrcType := Int" } GE_Contact(in1 := "CELLA", in2 := 230)
      { S7_Templates := "SrcType := DInt"; S7_Expression := "((IN1-IN2)*IN3)/IN4" } Calculate(in1 := "CELLA", in2 := 230, in3 := 1000, in4 := 245, out => "DB322_APP".IN12)
   END_RUNG
   RUNG wire#w1
      { S7_Templates := "SrcType := Int" } LT_Contact(in1 := "CELLA", in2 := 230)
      Move(in := 0, out1 => "DB322_APP".IN12)
   END_RUNG
   // the same network as SCL:
   IF "On" AND NOT "On" THEN
       "DB322_APP".IN10 := "CELLA";
       "DB322_APP".IN11 := "DB215_ProgramData".Offset_cella;
   END_IF;
   IF "On" AND ("CELLA" >= 230) THEN "DB322_APP".IN12 := (("CELLA"-230)*1000)/245; END_IF;
   IF "On" AND ("CELLA" < 230) THEN "DB322_APP".IN12 := 0; END_IF;
END_REGION

REGION Network 10: CALCOLO RIFERIMENTO CELLA SCALATO SU 255
   // "DB321_PID_M20".PID.M20_P08
   RUNG wire#powerrail
      Contact( "On" )
      wire#w1
      { S7_Templates := "SrcType := DInt"; S7_Expression := "(IN1*IN2-IN3)/IN4" } Calculate(in1 := "CELLA", in2 := 6765, in3 := 974690, in4 := 10000, out => #TempDint)
      I_Contact( "On" )
      { S7_Templates := "SrcType := DInt"; S7_Expression := "((IN1-IN2)*IN3/IN4)+IN5" } Calculate(in1 := "CELLA", in2 := "DB215_ProgramData".Offset_cella, in3 := 100, in4 := 317, in5 := 58, out => #TempDint_2)
   END_RUNG
   RUNG wire#w1
      Move(in := #TempDint, out1 => #TempInt)
   END_RUNG
   // the same network as SCL:
   IF "On" THEN #TempDint := ("CELLA"*6765-974690)/10000; END_IF;
   IF "On" AND NOT "On" THEN #TempDint_2 := (("CELLA"-"DB215_ProgramData".Offset_cella)*100/317)+58; END_IF;
   IF "On" THEN #TempInt := #TempDint; END_IF;
END_REGION

REGION Network 11: M20
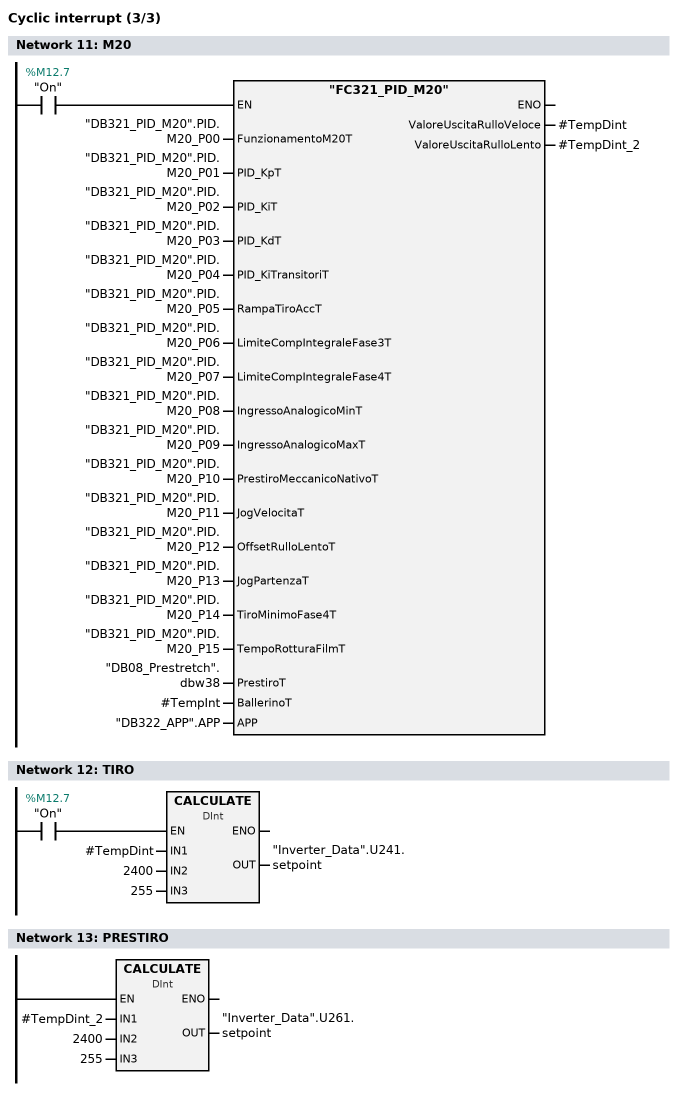
   RUNG wire#powerrail
      Contact( "On" )
      "FC321_PID_M20"(FunzionamentoM20T := "DB321_PID_M20".PID.M20_P00, PID_KpT := "DB321_PID_M20".PID.M20_P01, PID_KiT := "DB321_PID_M20".PID.M20_P02, PID_KdT := "DB321_PID_M20".PID.M20_P03, PID_KiTransitoriT := "DB321_PID_M20".PID.M20_P04, RampaTiroAccT := "DB321_PID_M20".PID.M20_P05, LimiteCompIntegraleFase3T := "DB321_PID_M20".PID.M20_P06, LimiteCompIntegraleFase4T := "DB321_PID_M20".PID.M20_P07, IngressoAnalogicoMinT := "DB321_PID_M20".PID.M20_P08, IngressoAnalogicoMaxT := "DB321_PID_M20".PID.M20_P09, PrestiroMeccanicoNativoT := "DB321_PID_M20".PID.M20_P10, JogVelocitaT := "DB321_PID_M20".PID.M20_P11, OffsetRulloLentoT := "DB321_PID_M20".PID.M20_P12, JogPartenzaT := "DB321_PID_M20".PID.M20_P13, TiroMinimoFase4T := "DB321_PID_M20".PID.M20_P14, TempoRotturaFilmT := "DB321_PID_M20".PID.M20_P15, PrestiroT := "DB08_Prestretch".dbw38, BallerinoT := #TempInt, APP := "DB322_APP".APP, ValoreUscitaRulloVeloce => #TempDint, ValoreUscitaRulloLento => #TempDint_2)
   END_RUNG
   // the same network as SCL:
   IF "On" THEN
       "FC321_PID_M20"(FunzionamentoM20T := "DB321_PID_M20".PID.M20_P00,
                       PID_KpT := "DB321_PID_M20".PID.M20_P01,
                       PID_KiT := "DB321_PID_M20".PID.M20_P02,
                       PID_KdT := "DB321_PID_M20".PID.M20_P03,
                       PID_KiTransitoriT := "DB321_PID_M20".PID.M20_P04,
                       RampaTiroAccT := "DB321_PID_M20".PID.M20_P05,
                       LimiteCompIntegraleFase3T := "DB321_PID_M20".PID.M20_P06,
                       LimiteCompIntegraleFase4T := "DB321_PID_M20".PID.M20_P07,
                       IngressoAnalogicoMinT := "DB321_PID_M20".PID.M20_P08,
                       IngressoAnalogicoMaxT := "DB321_PID_M20".PID.M20_P09,
                       PrestiroMeccanicoNativoT := "DB321_PID_M20".PID.M20_P10,
                       JogVelocitaT := "DB321_PID_M20".PID.M20_P11,
                       OffsetRulloLentoT := "DB321_PID_M20".PID.M20_P12,
                       JogPartenzaT := "DB321_PID_M20".PID.M20_P13,
                       TiroMinimoFase4T := "DB321_PID_M20".PID.M20_P14,
                       TempoRotturaFilmT := "DB321_PID_M20".PID.M20_P15,
                       PrestiroT := "DB08_Prestretch".dbw38,
                       BallerinoT := #TempInt,
                       APP := "DB322_APP".APP,
                       ValoreUscitaRulloVeloce => #TempDint,
                       ValoreUscitaRulloLento => #TempDint_2);
   END_IF;
END_REGION

REGION Network 12: TIRO
   RUNG wire#powerrail
      Contact( "On" )
      { S7_Templates := "SrcType := DInt"; S7_Expression := "IN1*IN2/IN3" } Calculate(in1 := #TempDint, in2 := 2400, in3 := 255, out => "Inverter_Data".U241.setpoint)
   END_RUNG
   // the same network as SCL:
   IF "On" THEN "Inverter_Data".U241.setpoint := #TempDint*2400/255; END_IF;
END_REGION

REGION Network 13: PRESTIRO
   RUNG wire#powerrail
      { S7_Templates := "SrcType := DInt"; S7_Expression := "IN1*IN2/IN3" } Calculate(in1 := #TempDint_2, in2 := 2400, in3 := 255, out => "Inverter_Data".U261.setpoint)
   END_RUNG
   // the same network as SCL:
   "Inverter_Data".U261.setpoint := #TempDint_2*2400/255;
END_REGION
END_ORGANIZATION_BLOCK

ORGANIZATION_BLOCK "Startup"   // OB100, LAD, Startup
TITLE = "Complete Restart"
{ S7_Optimized_Access := 'TRUE' }
VERSION : 0.1
// stored: AutoNumber false, IsIECCheckEnabled false, SetENOAutomatically false
   VAR_INPUT
      LostRetentive : Bool;   // True if retentive data are lost
      LostRTC : Bool;   // True if date and time are lost
   END_VAR
BEGIN

REGION Network 1: First cycle
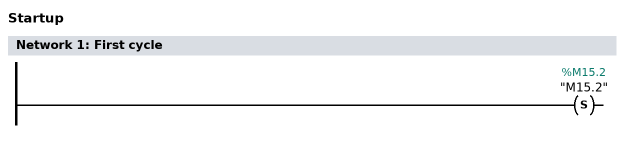
   RUNG wire#powerrail
      S_Coil( "M15.2" )
   END_RUNG
   // the same network as SCL:
   "M15.2" := TRUE;
END_REGION
END_ORGANIZATION_BLOCK

FUNCTION "FC101_AxisPositioningRev" : Void   // FC101, LAD
TITLE = Axis positioning
{ S7_Optimized_Access := 'FALSE' }
AUTHOR : Robopac
VERSION : 0.0
// stored: AutoNumber false, IsIECCheckEnabled false, SetENOAutomatically false, UDAEnableTagReadback false
   VAR_INPUT
      Start : Bool;   // Start dell'asse
      ExtraAvanti : Bool;   // Sensore di extracorsa avanti
      ExtraIndietro : Bool;   // Sensore di extracorsa indietro
      PosAttuale : Int;   // Posizione attuale dell'asse
      PosDest : Int;   // Posizione di destinazione dell'asse
      Dec : Int;   // Decelerazione
      H_Isteresi : Int;   // Isteresi
   END_VAR
   VAR_OUTPUT
      VelBassa : Bool;   // Asse all'interno dell'intervallo di decelerazione
      Avanti : Bool;   // Asse avanti
      Indietro : Bool;   // Asse indietro
   END_VAR
   VAR_IN_OUT
      PosOk : Bool;   // Asse in posizione
   END_VAR
   VAR_TEMP
      PosDestMenoH : Int;   // Posizione di destinazione asse-Isteresi
      PosDestPiuH : Int;   // Posizione di destinazione asse+Isteresi
      PosDestMenoDec : Int;   // Posizione di destinazione asse-Decelerazione
      PosDestPiuDec : Int;   // Posizione di destinazione asse+Decelerazione
   END_VAR
   VAR_TEMP   // added for the SCL form of the ladder/FBD networks
      _w1 : Bool;
   END_VAR
BEGIN

REGION Network 1
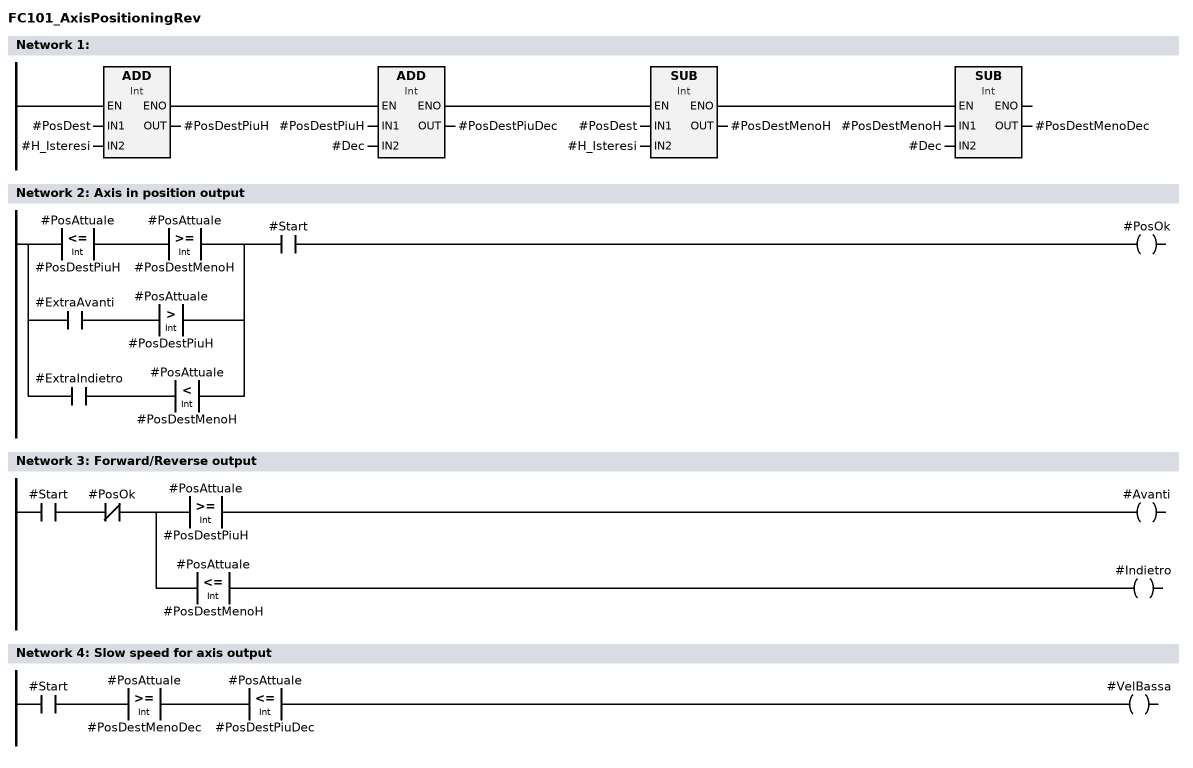
   RUNG wire#powerrail
      { S7_Templates := "SrcType := Int"; S7_GenerateENO := "TRUE" } Add(in1 := #PosDest, in2 := #H_Isteresi, out => #PosDestPiuH)
      { S7_Templates := "SrcType := Int"; S7_GenerateENO := "TRUE" } Add(in1 := #PosDestPiuH, in2 := #Dec, out => #PosDestPiuDec)
      { S7_Templates := "SrcType := Int"; S7_GenerateENO := "TRUE" } Sub(in1 := #PosDest, in2 := #H_Isteresi, out => #PosDestMenoH)
      { S7_Templates := "SrcType := Int"; S7_GenerateENO := "TRUE" } Sub(in1 := #PosDestMenoH, in2 := #Dec, out => #PosDestMenoDec)
   END_RUNG
   // the same network as SCL:
   // ENO of a box is taken as its EN; it also drops when the box reports an error
   #PosDestPiuH := #PosDest + #H_Isteresi;
   #PosDestPiuDec := #PosDestPiuH + #Dec;
   #PosDestMenoH := #PosDest - #H_Isteresi;
   #PosDestMenoDec := #PosDestMenoH - #Dec;
END_REGION

REGION Network 2: Axis in position output
   RUNG wire#powerrail
      { S7_Templates := "SrcType := Int" } LE_Contact(in1 := #PosAttuale, in2 := #PosDestPiuH)
      { S7_Templates := "SrcType := Int" } GE_Contact(in1 := #PosAttuale, in2 := #PosDestMenoH)
      wire#w1
      Contact( #Start )
      Coil( #PosOk )
   END_RUNG
   RUNG wire#powerrail
      Contact( #ExtraAvanti )
      { S7_Templates := "SrcType := Int" } GT_Contact(in1 := #PosAttuale, in2 := #PosDestPiuH)
   END_RUNG wire#w1
   RUNG wire#powerrail
      Contact( #ExtraIndietro )
      { S7_Templates := "SrcType := Int" } LT_Contact(in1 := #PosAttuale, in2 := #PosDestMenoH)
   END_RUNG wire#w1
   // the same network as SCL:
   #PosOk := (((#PosAttuale <= #PosDestPiuH) AND (#PosAttuale >= #PosDestMenoH)) OR (#ExtraAvanti AND (#PosAttuale > #PosDestPiuH)) OR (#ExtraIndietro AND (#PosAttuale < #PosDestMenoH))) AND #Start;
END_REGION

REGION Network 3: Forward/Reverse output
   RUNG wire#powerrail
      Contact( #Start )
      I_Contact( #PosOk )
      wire#w1
      { S7_Templates := "SrcType := Int" } GE_Contact(in1 := #PosAttuale, in2 := #PosDestPiuH)
      Coil( #Avanti )
   END_RUNG
   RUNG wire#w1
      { S7_Templates := "SrcType := Int" } LE_Contact(in1 := #PosAttuale, in2 := #PosDestMenoH)
      Coil( #Indietro )
   END_RUNG
   // the same network as SCL:
   #_w1 := #Start AND NOT #PosOk;
   #Avanti := #_w1 AND (#PosAttuale >= #PosDestPiuH);
   #Indietro := #_w1 AND (#PosAttuale <= #PosDestMenoH);
END_REGION

REGION Network 4: Slow speed for axis output
   RUNG wire#powerrail
      Contact( #Start )
      { S7_Templates := "SrcType := Int" } GE_Contact(in1 := #PosAttuale, in2 := #PosDestMenoDec)
      { S7_Templates := "SrcType := Int" } LE_Contact(in1 := #PosAttuale, in2 := #PosDestPiuDec)
      Coil( #VelBassa )
   END_RUNG
   // the same network as SCL:
   #VelBassa := #Start AND (#PosAttuale >= #PosDestMenoDec) AND (#PosAttuale <= #PosDestPiuDec);
END_REGION
END_FUNCTION

FUNCTION "FC38_DisplayEsaVT505" : Void   // FC38, LAD
TITLE = Display ESA VT505 management
{ S7_Optimized_Access := 'FALSE' }
AUTHOR : Robopac
VERSION : 0.0
// stored: AutoNumber false, IsIECCheckEnabled false, SetENOAutomatically false, UDAEnableTagReadback false
   VAR_TEMP
      TempInt : Int;
   END_VAR
   VAR_TEMP   // added for the SCL form of the ladder/FBD networks
      _w1 : Bool;
      _w2 : Bool;
      _w3 : Bool;
      _w4 : Bool;
      _w5 : Bool;
   END_VAR
BEGIN

REGION Network 1: Manual(Toggle bit): Pressure plate upward/downward (Helix)
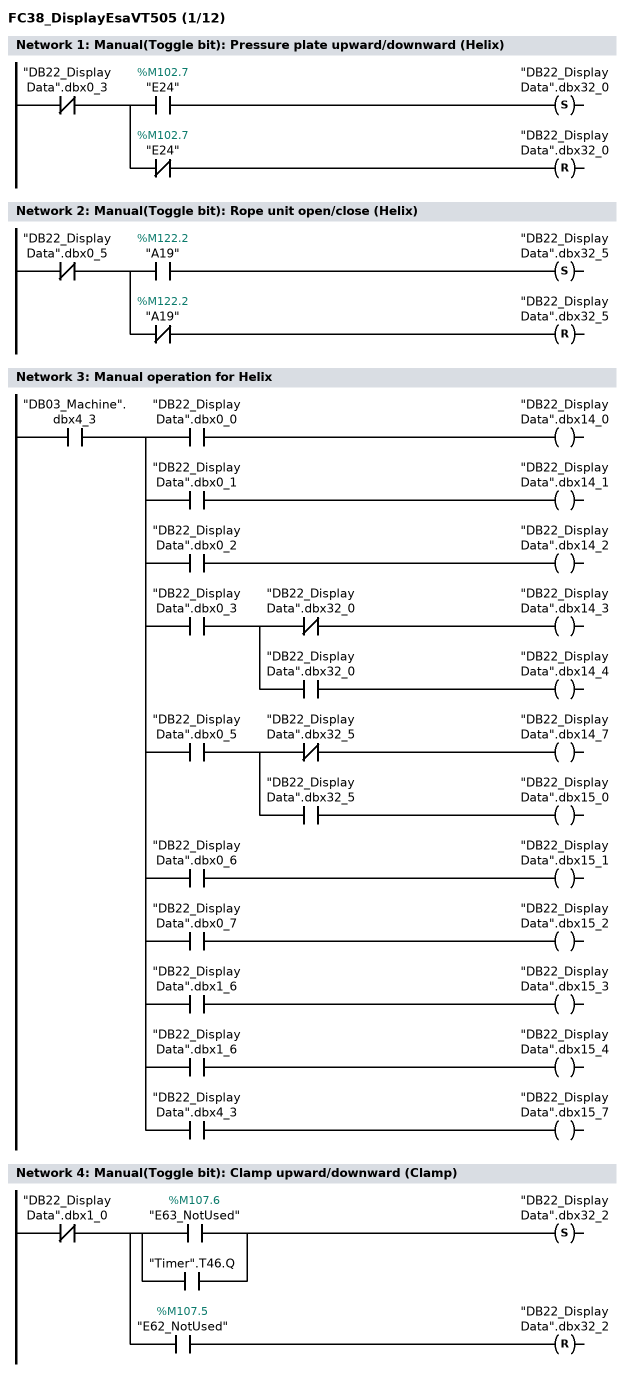
   RUNG wire#powerrail
      I_Contact( "DB22_DisplayData".dbx0_3 )
      wire#w1
      Contact( "E24" )
      S_Coil( "DB22_DisplayData".dbx32_0 )
   END_RUNG
   RUNG wire#w1
      I_Contact( "E24" )
      R_Coil( "DB22_DisplayData".dbx32_0 )
   END_RUNG
   // the same network as SCL:
   #_w1 := NOT "DB22_DisplayData".dbx0_3;
   IF #_w1 AND "E24" THEN "DB22_DisplayData".dbx32_0 := TRUE; END_IF;
   IF #_w1 AND NOT "E24" THEN "DB22_DisplayData".dbx32_0 := FALSE; END_IF;
END_REGION

REGION Network 2: Manual(Toggle bit): Rope unit open/close (Helix)
   RUNG wire#powerrail
      I_Contact( "DB22_DisplayData".dbx0_5 )
      wire#w1
      Contact( "A19" )
      S_Coil( "DB22_DisplayData".dbx32_5 )
   END_RUNG
   RUNG wire#w1
      I_Contact( "A19" )
      R_Coil( "DB22_DisplayData".dbx32_5 )
   END_RUNG
   // the same network as SCL:
   #_w1 := NOT "DB22_DisplayData".dbx0_5;
   IF #_w1 AND "A19" THEN "DB22_DisplayData".dbx32_5 := TRUE; END_IF;
   IF #_w1 AND NOT "A19" THEN "DB22_DisplayData".dbx32_5 := FALSE; END_IF;
END_REGION

REGION Network 3: Manual operation for Helix
   RUNG wire#powerrail
      Contact( "DB03_Machine".dbx4_3 )
      wire#w1
      Contact( "DB22_DisplayData".dbx0_0 )
      Coil( "DB22_DisplayData".dbx14_0 )
   END_RUNG
   RUNG wire#w1
      Contact( "DB22_DisplayData".dbx0_1 )
      Coil( "DB22_DisplayData".dbx14_1 )
   END_RUNG
   RUNG wire#w1
      Contact( "DB22_DisplayData".dbx0_2 )
      Coil( "DB22_DisplayData".dbx14_2 )
   END_RUNG
   RUNG wire#w1
      Contact( "DB22_DisplayData".dbx0_3 )
      wire#w2
      I_Contact( "DB22_DisplayData".dbx32_0 )
      Coil( "DB22_DisplayData".dbx14_3 )
   END_RUNG
   RUNG wire#w2
      Contact( "DB22_DisplayData".dbx32_0 )
      Coil( "DB22_DisplayData".dbx14_4 )
   END_RUNG
   RUNG wire#w1
      Contact( "DB22_DisplayData".dbx0_5 )
      wire#w3
      I_Contact( "DB22_DisplayData".dbx32_5 )
      Coil( "DB22_DisplayData".dbx14_7 )
   END_RUNG
   RUNG wire#w3
      Contact( "DB22_DisplayData".dbx32_5 )
      Coil( "DB22_DisplayData".dbx15_0 )
   END_RUNG
   RUNG wire#w1
      Contact( "DB22_DisplayData".dbx0_6 )
      Coil( "DB22_DisplayData".dbx15_1 )
   END_RUNG
   RUNG wire#w1
      Contact( "DB22_DisplayData".dbx0_7 )
      Coil( "DB22_DisplayData".dbx15_2 )
   END_RUNG
   RUNG wire#w1
      Contact( "DB22_DisplayData".dbx1_6 )
      Coil( "DB22_DisplayData".dbx15_3 )
   END_RUNG
   RUNG wire#w1
      Contact( "DB22_DisplayData".dbx1_6 )
      Coil( "DB22_DisplayData".dbx15_4 )
   END_RUNG
   RUNG wire#w1
      Contact( "DB22_DisplayData".dbx4_3 )
      Coil( "DB22_DisplayData".dbx15_7 )
   END_RUNG
   // the same network as SCL:
   "DB22_DisplayData".dbx14_0 := "DB03_Machine".dbx4_3 AND "DB22_DisplayData".dbx0_0;
   "DB22_DisplayData".dbx14_1 := "DB03_Machine".dbx4_3 AND "DB22_DisplayData".dbx0_1;
   "DB22_DisplayData".dbx14_2 := "DB03_Machine".dbx4_3 AND "DB22_DisplayData".dbx0_2;
   #_w1 := "DB03_Machine".dbx4_3 AND "DB22_DisplayData".dbx0_3;
   "DB22_DisplayData".dbx14_3 := #_w1 AND NOT "DB22_DisplayData".dbx32_0;
   "DB22_DisplayData".dbx14_4 := #_w1 AND "DB22_DisplayData".dbx32_0;
   #_w2 := "DB03_Machine".dbx4_3 AND "DB22_DisplayData".dbx0_5;
   "DB22_DisplayData".dbx14_7 := #_w2 AND NOT "DB22_DisplayData".dbx32_5;
   "DB22_DisplayData".dbx15_0 := #_w2 AND "DB22_DisplayData".dbx32_5;
   "DB22_DisplayData".dbx15_1 := "DB03_Machine".dbx4_3 AND "DB22_DisplayData".dbx0_6;
   "DB22_DisplayData".dbx15_2 := "DB03_Machine".dbx4_3 AND "DB22_DisplayData".dbx0_7;
   "DB22_DisplayData".dbx15_3 := "DB03_Machine".dbx4_3 AND "DB22_DisplayData".dbx1_6;
   "DB22_DisplayData".dbx15_4 := "DB03_Machine".dbx4_3 AND "DB22_DisplayData".dbx1_6;
   "DB22_DisplayData".dbx15_7 := "DB03_Machine".dbx4_3 AND "DB22_DisplayData".dbx4_3;
END_REGION

REGION Network 4: Manual(Toggle bit): Clamp upward/downward (Clamp)
   RUNG wire#powerrail
      I_Contact( "DB22_DisplayData".dbx1_0 )
      wire#w1
      Contact( "E63_NotUsed" )
      wire#w2
      S_Coil( "DB22_DisplayData".dbx32_2 )
   END_RUNG
   RUNG wire#w1
      Contact( "Timer".T46.Q )
   END_RUNG wire#w2
   RUNG wire#w1
      Contact( "E62_NotUsed" )
      R_Coil( "DB22_DisplayData".dbx32_2 )
   END_RUNG
   // the same network as SCL:
   #_w1 := NOT "DB22_DisplayData".dbx1_0;
   IF #_w1 AND ("E63_NotUsed" OR "Timer".T46.Q) THEN "DB22_DisplayData".dbx32_2 := TRUE; END_IF;
   IF #_w1 AND "E62_NotUsed" THEN "DB22_DisplayData".dbx32_2 := FALSE; END_IF;
END_REGION

REGION Network 5: Manual(Toggle bit): Welder unit upward/downward (Clamp)
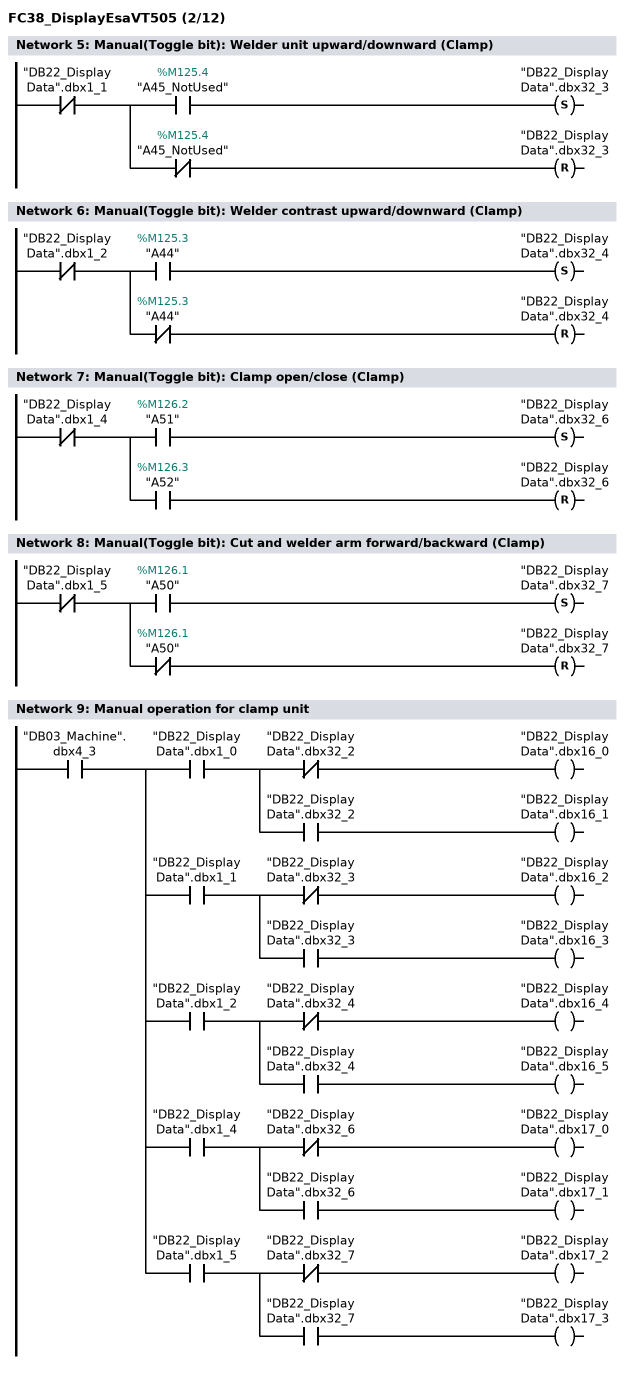
   RUNG wire#powerrail
      I_Contact( "DB22_DisplayData".dbx1_1 )
      wire#w1
      Contact( "A45_NotUsed" )
      S_Coil( "DB22_DisplayData".dbx32_3 )
   END_RUNG
   RUNG wire#w1
      I_Contact( "A45_NotUsed" )
      R_Coil( "DB22_DisplayData".dbx32_3 )
   END_RUNG
   // the same network as SCL:
   #_w1 := NOT "DB22_DisplayData".dbx1_1;
   IF #_w1 AND "A45_NotUsed" THEN "DB22_DisplayData".dbx32_3 := TRUE; END_IF;
   IF #_w1 AND NOT "A45_NotUsed" THEN "DB22_DisplayData".dbx32_3 := FALSE; END_IF;
END_REGION

REGION Network 6: Manual(Toggle bit): Welder contrast upward/downward (Clamp)
   RUNG wire#powerrail
      I_Contact( "DB22_DisplayData".dbx1_2 )
      wire#w1
      Contact( "A44" )
      S_Coil( "DB22_DisplayData".dbx32_4 )
   END_RUNG
   RUNG wire#w1
      I_Contact( "A44" )
      R_Coil( "DB22_DisplayData".dbx32_4 )
   END_RUNG
   // the same network as SCL:
   #_w1 := NOT "DB22_DisplayData".dbx1_2;
   IF #_w1 AND "A44" THEN "DB22_DisplayData".dbx32_4 := TRUE; END_IF;
   IF #_w1 AND NOT "A44" THEN "DB22_DisplayData".dbx32_4 := FALSE; END_IF;
END_REGION

REGION Network 7: Manual(Toggle bit): Clamp open/close (Clamp)
   RUNG wire#powerrail
      I_Contact( "DB22_DisplayData".dbx1_4 )
      wire#w1
      Contact( "A51" )
      S_Coil( "DB22_DisplayData".dbx32_6 )
   END_RUNG
   RUNG wire#w1
      Contact( "A52" )
      R_Coil( "DB22_DisplayData".dbx32_6 )
   END_RUNG
   // the same network as SCL:
   #_w1 := NOT "DB22_DisplayData".dbx1_4;
   IF #_w1 AND "A51" THEN "DB22_DisplayData".dbx32_6 := TRUE; END_IF;
   IF #_w1 AND "A52" THEN "DB22_DisplayData".dbx32_6 := FALSE; END_IF;
END_REGION

REGION Network 8: Manual(Toggle bit): Cut and welder arm forward/backward (Clamp)
   RUNG wire#powerrail
      I_Contact( "DB22_DisplayData".dbx1_5 )
      wire#w1
      Contact( "A50" )
      S_Coil( "DB22_DisplayData".dbx32_7 )
   END_RUNG
   RUNG wire#w1
      I_Contact( "A50" )
      R_Coil( "DB22_DisplayData".dbx32_7 )
   END_RUNG
   // the same network as SCL:
   #_w1 := NOT "DB22_DisplayData".dbx1_5;
   IF #_w1 AND "A50" THEN "DB22_DisplayData".dbx32_7 := TRUE; END_IF;
   IF #_w1 AND NOT "A50" THEN "DB22_DisplayData".dbx32_7 := FALSE; END_IF;
END_REGION

REGION Network 9: Manual operation for clamp unit
   RUNG wire#powerrail
      Contact( "DB03_Machine".dbx4_3 )
      wire#w1
      Contact( "DB22_DisplayData".dbx1_0 )
      wire#w2
      I_Contact( "DB22_DisplayData".dbx32_2 )
      Coil( "DB22_DisplayData".dbx16_0 )
   END_RUNG
   RUNG wire#w2
      Contact( "DB22_DisplayData".dbx32_2 )
      Coil( "DB22_DisplayData".dbx16_1 )
   END_RUNG
   RUNG wire#w1
      Contact( "DB22_DisplayData".dbx1_1 )
      wire#w3
      I_Contact( "DB22_DisplayData".dbx32_3 )
      Coil( "DB22_DisplayData".dbx16_2 )
   END_RUNG
   RUNG wire#w3
      Contact( "DB22_DisplayData".dbx32_3 )
      Coil( "DB22_DisplayData".dbx16_3 )
   END_RUNG
   RUNG wire#w1
      Contact( "DB22_DisplayData".dbx1_2 )
      wire#w4
      I_Contact( "DB22_DisplayData".dbx32_4 )
      Coil( "DB22_DisplayData".dbx16_4 )
   END_RUNG
   RUNG wire#w4
      Contact( "DB22_DisplayData".dbx32_4 )
      Coil( "DB22_DisplayData".dbx16_5 )
   END_RUNG
   RUNG wire#w1
      Contact( "DB22_DisplayData".dbx1_4 )
      wire#w5
      I_Contact( "DB22_DisplayData".dbx32_6 )
      Coil( "DB22_DisplayData".dbx17_0 )
   END_RUNG
   RUNG wire#w5
      Contact( "DB22_DisplayData".dbx32_6 )
      Coil( "DB22_DisplayData".dbx17_1 )
   END_RUNG
   RUNG wire#w1
      Contact( "DB22_DisplayData".dbx1_5 )
      wire#w6
      I_Contact( "DB22_DisplayData".dbx32_7 )
      Coil( "DB22_DisplayData".dbx17_2 )
   END_RUNG
   RUNG wire#w6
      Contact( "DB22_DisplayData".dbx32_7 )
      Coil( "DB22_DisplayData".dbx17_3 )
   END_RUNG
   // the same network as SCL:
   #_w1 := "DB03_Machine".dbx4_3 AND "DB22_DisplayData".dbx1_0;
   "DB22_DisplayData".dbx16_0 := #_w1 AND NOT "DB22_DisplayData".dbx32_2;
   "DB22_DisplayData".dbx16_1 := #_w1 AND "DB22_DisplayData".dbx32_2;
   #_w2 := "DB03_Machine".dbx4_3 AND "DB22_DisplayData".dbx1_1;
   "DB22_DisplayData".dbx16_2 := #_w2 AND NOT "DB22_DisplayData".dbx32_3;
   "DB22_DisplayData".dbx16_3 := #_w2 AND "DB22_DisplayData".dbx32_3;
   #_w3 := "DB03_Machine".dbx4_3 AND "DB22_DisplayData".dbx1_2;
   "DB22_DisplayData".dbx16_4 := #_w3 AND NOT "DB22_DisplayData".dbx32_4;
   "DB22_DisplayData".dbx16_5 := #_w3 AND "DB22_DisplayData".dbx32_4;
   #_w4 := "DB03_Machine".dbx4_3 AND "DB22_DisplayData".dbx1_4;
   "DB22_DisplayData".dbx17_0 := #_w4 AND NOT "DB22_DisplayData".dbx32_6;
   "DB22_DisplayData".dbx17_1 := #_w4 AND "DB22_DisplayData".dbx32_6;
   #_w5 := "DB03_Machine".dbx4_3 AND "DB22_DisplayData".dbx1_5;
   "DB22_DisplayData".dbx17_2 := #_w5 AND NOT "DB22_DisplayData".dbx32_7;
   "DB22_DisplayData".dbx17_3 := #_w5 AND "DB22_DisplayData".dbx32_7;
END_REGION

REGION Network 10: Manual(Toggle bit): Opening/closing clamp to pull top film (Top)
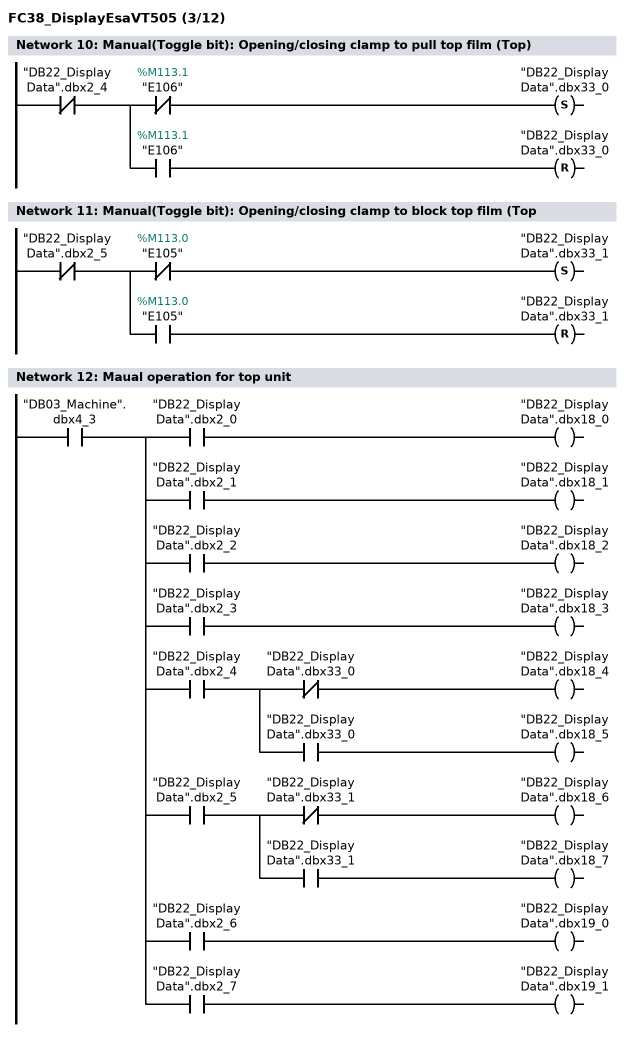
   RUNG wire#powerrail
      I_Contact( "DB22_DisplayData".dbx2_4 )
      wire#w1
      I_Contact( "E106" )
      S_Coil( "DB22_DisplayData".dbx33_0 )
   END_RUNG
   RUNG wire#w1
      Contact( "E106" )
      R_Coil( "DB22_DisplayData".dbx33_0 )
   END_RUNG
   // the same network as SCL:
   #_w1 := NOT "DB22_DisplayData".dbx2_4;
   IF #_w1 AND NOT "E106" THEN "DB22_DisplayData".dbx33_0 := TRUE; END_IF;
   IF #_w1 AND "E106" THEN "DB22_DisplayData".dbx33_0 := FALSE; END_IF;
END_REGION

REGION Network 11: Manual(Toggle bit): Opening/closing clamp to block top film (Top
   RUNG wire#powerrail
      I_Contact( "DB22_DisplayData".dbx2_5 )
      wire#w1
      I_Contact( "E105" )
      S_Coil( "DB22_DisplayData".dbx33_1 )
   END_RUNG
   RUNG wire#w1
      Contact( "E105" )
      R_Coil( "DB22_DisplayData".dbx33_1 )
   END_RUNG
   // the same network as SCL:
   #_w1 := NOT "DB22_DisplayData".dbx2_5;
   IF #_w1 AND NOT "E105" THEN "DB22_DisplayData".dbx33_1 := TRUE; END_IF;
   IF #_w1 AND "E105" THEN "DB22_DisplayData".dbx33_1 := FALSE; END_IF;
END_REGION

REGION Network 12: Maual operation for top unit
   RUNG wire#powerrail
      Contact( "DB03_Machine".dbx4_3 )
      wire#w1
      Contact( "DB22_DisplayData".dbx2_0 )
      Coil( "DB22_DisplayData".dbx18_0 )
   END_RUNG
   RUNG wire#w1
      Contact( "DB22_DisplayData".dbx2_1 )
      Coil( "DB22_DisplayData".dbx18_1 )
   END_RUNG
   RUNG wire#w1
      Contact( "DB22_DisplayData".dbx2_2 )
      Coil( "DB22_DisplayData".dbx18_2 )
   END_RUNG
   RUNG wire#w1
      Contact( "DB22_DisplayData".dbx2_3 )
      Coil( "DB22_DisplayData".dbx18_3 )
   END_RUNG
   RUNG wire#w1
      Contact( "DB22_DisplayData".dbx2_4 )
      wire#w2
      I_Contact( "DB22_DisplayData".dbx33_0 )
      Coil( "DB22_DisplayData".dbx18_4 )
   END_RUNG
   RUNG wire#w2
      Contact( "DB22_DisplayData".dbx33_0 )
      Coil( "DB22_DisplayData".dbx18_5 )
   END_RUNG
   RUNG wire#w1
      Contact( "DB22_DisplayData".dbx2_5 )
      wire#w3
      I_Contact( "DB22_DisplayData".dbx33_1 )
      Coil( "DB22_DisplayData".dbx18_6 )
   END_RUNG
   RUNG wire#w3
      Contact( "DB22_DisplayData".dbx33_1 )
      Coil( "DB22_DisplayData".dbx18_7 )
   END_RUNG
   RUNG wire#w1
      Contact( "DB22_DisplayData".dbx2_6 )
      Coil( "DB22_DisplayData".dbx19_0 )
   END_RUNG
   RUNG wire#w1
      Contact( "DB22_DisplayData".dbx2_7 )
      Coil( "DB22_DisplayData".dbx19_1 )
   END_RUNG
   // the same network as SCL:
   "DB22_DisplayData".dbx18_0 := "DB03_Machine".dbx4_3 AND "DB22_DisplayData".dbx2_0;
   "DB22_DisplayData".dbx18_1 := "DB03_Machine".dbx4_3 AND "DB22_DisplayData".dbx2_1;
   "DB22_DisplayData".dbx18_2 := "DB03_Machine".dbx4_3 AND "DB22_DisplayData".dbx2_2;
   "DB22_DisplayData".dbx18_3 := "DB03_Machine".dbx4_3 AND "DB22_DisplayData".dbx2_3;
   #_w1 := "DB03_Machine".dbx4_3 AND "DB22_DisplayData".dbx2_4;
   "DB22_DisplayData".dbx18_4 := #_w1 AND NOT "DB22_DisplayData".dbx33_0;
   "DB22_DisplayData".dbx18_5 := #_w1 AND "DB22_DisplayData".dbx33_0;
   #_w2 := "DB03_Machine".dbx4_3 AND "DB22_DisplayData".dbx2_5;
   "DB22_DisplayData".dbx18_6 := #_w2 AND NOT "DB22_DisplayData".dbx33_1;
   "DB22_DisplayData".dbx18_7 := #_w2 AND "DB22_DisplayData".dbx33_1;
   "DB22_DisplayData".dbx19_0 := "DB03_Machine".dbx4_3 AND "DB22_DisplayData".dbx2_6;
   "DB22_DisplayData".dbx19_1 := "DB03_Machine".dbx4_3 AND "DB22_DisplayData".dbx2_7;
END_REGION

REGION Network 13: Diagnostic signal conveyor
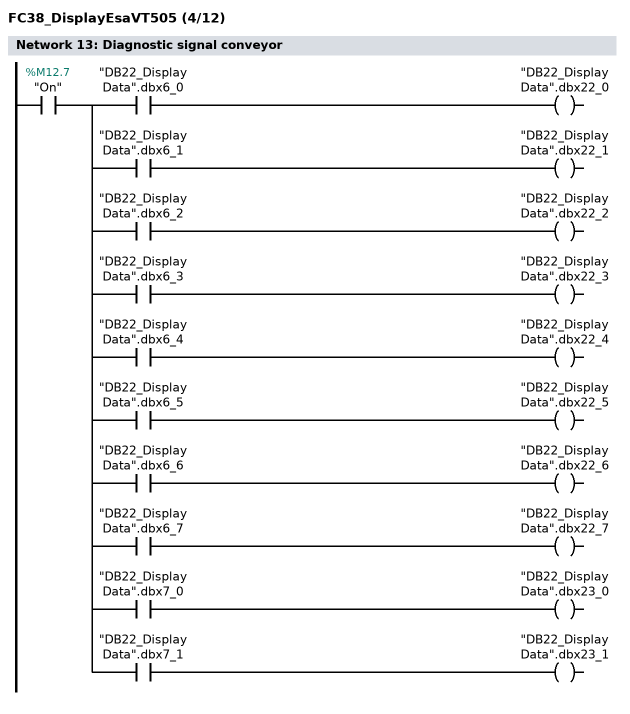
   RUNG wire#powerrail
      Contact( "On" )
      wire#w1
      Contact( "DB22_DisplayData".dbx6_0 )
      Coil( "DB22_DisplayData".dbx22_0 )
   END_RUNG
   RUNG wire#w1
      Contact( "DB22_DisplayData".dbx6_1 )
      Coil( "DB22_DisplayData".dbx22_1 )
   END_RUNG
   RUNG wire#w1
      Contact( "DB22_DisplayData".dbx6_2 )
      Coil( "DB22_DisplayData".dbx22_2 )
   END_RUNG
   RUNG wire#w1
      Contact( "DB22_DisplayData".dbx6_3 )
      Coil( "DB22_DisplayData".dbx22_3 )
   END_RUNG
   RUNG wire#w1
      Contact( "DB22_DisplayData".dbx6_4 )
      Coil( "DB22_DisplayData".dbx22_4 )
   END_RUNG
   RUNG wire#w1
      Contact( "DB22_DisplayData".dbx6_5 )
      Coil( "DB22_DisplayData".dbx22_5 )
   END_RUNG
   RUNG wire#w1
      Contact( "DB22_DisplayData".dbx6_6 )
      Coil( "DB22_DisplayData".dbx22_6 )
   END_RUNG
   RUNG wire#w1
      Contact( "DB22_DisplayData".dbx6_7 )
      Coil( "DB22_DisplayData".dbx22_7 )
   END_RUNG
   RUNG wire#w1
      Contact( "DB22_DisplayData".dbx7_0 )
      Coil( "DB22_DisplayData".dbx23_0 )
   END_RUNG
   RUNG wire#w1
      Contact( "DB22_DisplayData".dbx7_1 )
      Coil( "DB22_DisplayData".dbx23_1 )
   END_RUNG
   // the same network as SCL:
   "DB22_DisplayData".dbx22_0 := "On" AND "DB22_DisplayData".dbx6_0;
   "DB22_DisplayData".dbx22_1 := "On" AND "DB22_DisplayData".dbx6_1;
   "DB22_DisplayData".dbx22_2 := "On" AND "DB22_DisplayData".dbx6_2;
   "DB22_DisplayData".dbx22_3 := "On" AND "DB22_DisplayData".dbx6_3;
   "DB22_DisplayData".dbx22_4 := "On" AND "DB22_DisplayData".dbx6_4;
   "DB22_DisplayData".dbx22_5 := "On" AND "DB22_DisplayData".dbx6_5;
   "DB22_DisplayData".dbx22_6 := "On" AND "DB22_DisplayData".dbx6_6;
   "DB22_DisplayData".dbx22_7 := "On" AND "DB22_DisplayData".dbx6_7;
   "DB22_DisplayData".dbx23_0 := "On" AND "DB22_DisplayData".dbx7_0;
   "DB22_DisplayData".dbx23_1 := "On" AND "DB22_DisplayData".dbx7_1;
END_REGION

REGION Network 14: Diagnostic signal conveyor
